C03628=1105.080,205.450,-68.281,178.823,14.144,151.208
C03629=1105.087,205.699,-68.305,178.828,14.143,151.207
C03630=1105.092,205.948,-68.330,178.832,14.142,151.206
C03631=1105.098,206.197,-68.354,178.836,14.141,151.205
C03632=1105.103,206.446,-68.379,178.840,14.139,151.203
C03633=1105.109,206.694,-68.403,178.845,14.138,151.202
C03634=1105.115,206.943,-68.427,178.848,14.136,151.201
C03635=1105.121,207.191,-68.452,178.853,14.136,151.200
C03636=1105.126,207.440,-68.476,178.857,14.134,151.198
C03637=1105.132,207.689,-68.501,178.861,14.133,151.197
C03638=1105.156,208.685,-68.598,178.887,14.133,151.191
C03639=1105.163,209.052,-68.635,178.893,14.132,151.190
C03640=1105.171,209.419,-68.670,178.899,14.131,151.188
C03641=1105.181,209.786,-68.707,178.904,14.131,151.187
C03642=1105.189,210.152,-68.743,178.911,14.131,151.186
C03643=1105.195,210.402,-68.768,178.914,14.129,151.185
C03644=1105.200,210.650,-68.792,178.918,14.129,151.184
C03645=1105.206,210.899,-68.817,178.922,14.129,151.183
C03646=1105.211,211.147,-68.841,178.926,14.129,151.182
C03647=1105.217,211.397,-68.866,178.930,14.128,151.181
C03648=1105.223,211.645,-68.891,178.934,14.127,151.180
C03649=1105.228,211.893,-68.915,178.938,14.127,151.179
C03650=1105.234,212.143,-68.940,178.942,14.126,151.178
C03651=1105.240,212.390,-68.965,178.946,14.126,151.177
C03652=1105.246,212.640,-68.990,178.949,14.125,151.176
C03653=1105.251,212.888,-69.014,178.953,14.125,151.175
C03654=1105.256,213.137,-69.040,178.958,14.125,151.174
C03655=1105.262,213.386,-69.064,178.961,14.125,151.173
C03656=1105.268,213.635,-69.089,178.966,14.124,151.172
C03657=1105.273,213.883,-69.114,178.969,14.123,151.171
C03658=1105.279,214.132,-69.139,178.973,14.123,151.170
C03659=1105.285,214.381,-69.164,178.977,14.123,151.169
C03660=1105.291,214.629,-69.188,178.981,14.122,151.168
C03661=1105.296,214.879,-69.214,178.985,14.122,151.167
C03662=1105.302,215.127,-69.239,178.989,14.122,151.166
C03663=1105.308,215.376,-69.263,178.993,14.121,151.165
C03664=1105.313,215.624,-69.288,178.997,14.120,151.164
C03665=1105.319,215.873,-69.313,179.001,14.120,151.163
C03666=1105.325,216.121,-69.338,179.005,14.120,151.162
C03667=1105.330,216.371,-69.363,179.009,14.119,151.161
C03668=1105.335,216.619,-69.388,179.012,14.119,151.160
C03669=1105.341,216.868,-69.413,179.017,14.118,151.159
C03670=1105.348,217.117,-69.438,179.020,14.118,151.158
C03671=1105.352,217.365,-69.464,179.025,14.118,151.157
C03672=1105.358,217.614,-69.488,179.029,14.118,151.156
C03673=1105.364,217.862,-69.513,179.033,14.117,151.155
C03674=1105.370,218.111,-69.539,179.036,14.116,151.154
C03675=1105.375,218.361,-69.564,179.040,14.116,151.153
C03676=1105.381,218.608,-69.589,179.044,14.116,151.152
C03677=1105.387,218.857,-69.614,179.048,14.115,151.151
C03678=1105.392,219.106,-69.638,179.052,14.115,151.150
C03679=1105.398,219.355,-69.664,179.056,14.115,151.149
C03680=1105.404,219.603,-69.690,179.060,14.114,151.148
C03681=1105.409,219.852,-69.714,179.064,14.114,151.147
C03682=1105.415,220.101,-69.740,179.068,14.113,151.146
C03683=1105.421,220.350,-69.765,179.072,14.113,151.145
C03684=1105.427,220.598,-69.790,179.076,14.113,151.144
C03685=1105.433,220.847,-69.815,179.080,14.112,151.143
C03686=1105.438,221.096,-69.841,179.083,14.112,151.142
C03687=1105.444,221.344,-69.866,179.087,14.111,151.141
C03688=1105.450,221.592,-69.891,179.092,14.111,151.140
C03689=1105.455,221.841,-69.917,179.096,14.111,151.139
C03690=1105.461,222.089,-69.942,179.100,14.110,151.138
C03691=1105.470,222.460,-69.980,179.105,14.110,151.137
C03692=1105.477,222.831,-70.017,179.111,14.109,151.135
C03693=1105.486,223.201,-70.056,179.117,14.108,151.134
C03694=1105.494,223.571,-70.093,179.123,14.108,151.133
C03695=1105.501,223.820,-70.119,179.127,14.108,151.132
C03696=1105.506,224.068,-70.144,179.131,14.107,151.131
C03697=1105.512,224.316,-70.169,179.134,14.107,151.130
C03698=1105.517,224.565,-70.195,179.139,14.107,151.129
C03699=1105.523,224.814,-70.221,179.143,14.107,151.128
C03700=1105.528,225.062,-70.246,179.147,14.106,151.127
C03701=1105.534,225.311,-70.272,179.151,14.106,151.126
C03702=1105.540,225.560,-70.298,179.155,14.106,151.125
C03703=1105.545,225.808,-70.323,179.159,14.106,151.124
C03704=1105.551,226.057,-70.348,179.162,14.105,151.123
C03705=1105.556,226.306,-70.374,179.166,14.104,151.122
C03706=1105.563,226.555,-70.400,179.170,14.104,151.121
C03707=1105.568,226.804,-70.426,179.174,14.104,151.120
C03708=1105.574,227.052,-70.451,179.178,14.104,151.119
C03709=1105.579,227.301,-70.477,179.182,14.103,151.118
C03710=1105.585,227.549,-70.502,179.186,14.103,151.117
C03711=1105.591,227.798,-70.528,179.191,14.103,151.116
C03712=1105.596,228.047,-70.553,179.194,14.102,151.115
C03713=1105.602,228.295,-70.579,179.198,14.102,151.114
C03714=1105.608,228.544,-70.605,179.202,14.102,151.113
C03715=1105.614,228.792,-70.631,179.206,14.102,151.112
C03716=1105.619,229.041,-70.657,179.210,14.101,151.111
C03717=1105.625,229.290,-70.683,179.214,14.101,151.110
C03718=1105.631,229.538,-70.708,179.218,14.101,151.109
C03719=1105.636,229.787,-70.734,179.222,14.101,151.108
C03720=1105.642,230.035,-70.760,179.226,14.100,151.107
C03721=1105.648,230.284,-70.785,179.229,14.100,151.107
C03722=1105.654,230.533,-70.812,179.234,14.099,151.105
C03723=1105.659,230.782,-70.838,179.237,14.099,151.105
C03724=1105.665,231.030,-70.863,179.241,14.099,151.104
C03725=1105.670,231.278,-70.889,179.246,14.099,151.103
C03726=1105.676,231.527,-70.916,179.250,14.099,151.102
C03727=1105.682,231.776,-70.942,179.254,14.098,151.101
C03728=1105.688,232.024,-70.967,179.258,14.098,151.100
C03729=1105.693,232.273,-70.994,179.262,14.098,151.099
C03730=1105.699,232.522,-71.019,179.266,14.098,151.098
C03731=1105.704,232.771,-71.045,179.269,14.097,151.097
C03732=1105.710,233.018,-71.072,179.273,14.097,151.096
C03733=1105.716,233.267,-71.097,179.277,14.097,151.095
C03734=1105.722,233.515,-71.124,179.281,14.096,151.094
C03735=1105.727,233.764,-71.150,179.285,14.096,151.093
C03736=1105.733,234.013,-71.175,179.289,14.096,151.092
C03737=1105.738,234.262,-71.202,179.293,14.096,151.091
C03738=1105.744,234.510,-71.227,179.297,14.096,151.090
C03739=1105.750,234.759,-71.254,179.301,14.096,151.089
C03740=1105.756,235.008,-71.280,179.305,14.096,151.089
C03741=1105.762,235.256,-71.307,179.309,14.095,151.087
C03742=1105.766,235.504,-71.332,179.313,14.095,151.087
C03743=1105.775,235.867,-71.371,179.319,14.094,151.085
C03744=1105.783,236.228,-71.409,179.324,14.094,151.084
C03745=1105.791,236.590,-71.448,179.330,14.094,151.083
C03746=1105.799,236.952,-71.486,179.336,14.094,151.081
C03747=1105.805,237.201,-71.512,179.340,14.094,151.080
C03748=1105.810,237.449,-71.539,179.344,14.093,151.079
C03749=1105.816,237.698,-71.564,179.348,14.093,151.078
C03750=1105.822,237.946,-71.591,179.351,14.093,151.077
C03751=1105.828,238.194,-71.617,179.355,14.092,151.076
C03752=1105.834,238.443,-71.643,179.359,14.092,151.075
C03753=1105.839,238.692,-71.670,179.363,14.092,151.075
C03754=1105.845,238.940,-71.696,179.367,14.092,151.074
C03755=1105.851,239.189,-71.722,179.371,14.092,151.073
C03756=1105.856,239.437,-71.749,179.375,14.092,151.072
C03757=1105.862,239.686,-71.776,179.379,14.091,151.071
C03758=1105.868,239.935,-71.802,179.383,14.091,151.070
C03759=1105.874,240.183,-71.828,179.387,14.091,151.069
C03760=1105.879,240.432,-71.855,179.391,14.091,151.068
C03761=1105.884,240.680,-71.882,179.395,14.091,151.067
C03762=1105.890,240.929,-71.908,179.399,14.091,151.066
C03763=1105.896,241.178,-71.935,179.403,14.091,151.065
C03764=1105.902,241.426,-71.962,179.407,14.090,151.064
C03765=1105.908,241.675,-71.988,179.411,14.090,151.063
C03766=1105.913,241.923,-72.015,179.415,14.090,151.062
C03767=1105.919,242.172,-72.042,179.419,14.090,151.061
C03768=1105.925,242.420,-72.068,179.423,14.090,151.060
C03769=1105.931,242.669,-72.094,179.427,14.090,151.060
C03770=1105.936,242.917,-72.121,179.431,14.090,151.059
C03771=1105.942,243.166,-72.147,179.435,14.090,151.058
C03772=1105.947,243.414,-72.175,179.439,14.090,151.057
C03773=1105.953,243.663,-72.201,179.443,14.090,151.056
C03774=1105.959,243.911,-72.228,179.446,14.089,151.055
C03775=1105.964,244.159,-72.255,179.450,14.089,151.054
C03776=1105.970,244.409,-72.282,179.454,14.089,151.053
C03777=1105.976,244.657,-72.309,179.458,14.089,151.052
C03778=1105.982,244.905,-72.336,179.462,14.089,151.051
C03779=1105.987,245.154,-72.362,179.466,14.089,151.050
C03780=1105.992,245.402,-72.389,179.470,14.088,151.049
C03781=1105.998,245.651,-72.416,179.474,14.088,151.049
C03782=1106.004,245.899,-72.443,179.478,14.088,151.048
C03783=1106.010,246.148,-72.469,179.482,14.088,151.047
C03784=1106.015,246.396,-72.497,179.486,14.088,151.046
C03785=1106.021,246.645,-72.524,179.490,14.088,151.045
C03786=1106.027,246.894,-72.550,179.494,14.088,151.044
C03787=1106.032,247.142,-72.578,179.498,14.088,151.043
C03788=1106.038,247.391,-72.604,179.501,14.088,151.042
C03789=1106.043,247.639,-72.631,179.505,14.088,151.041
C03790=1106.049,247.888,-72.658,179.510,14.087,151.040
C03791=1106.055,248.135,-72.685,179.513,14.087,151.039
C03792=1106.060,248.384,-72.712,179.517,14.087,151.039
C03793=1106.066,248.633,-72.740,179.521,14.087,151.038
C03794=1106.072,248.882,-72.766,179.525,14.087,151.037
C03795=1106.079,249.237,-72.805,179.531,14.088,151.036
C03796=1106.087,249.591,-72.844,179.537,14.087,151.034
C03797=1106.095,249.947,-72.883,179.542,14.087,151.033
C03798=1106.104,250.302,-72.921,179.548,14.088,151.032
C03799=1106.109,250.550,-72.949,179.552,14.088,151.031
C03800=1106.115,250.799,-72.976,179.556,14.088,151.030
C03801=1106.120,251.047,-73.003,179.560,14.088,151.029
C03802=1106.127,251.296,-73.031,179.564,14.088,151.028
C03803=1106.132,251.544,-73.058,179.568,14.088,151.027
C03804=1106.137,251.793,-73.085,179.572,14.088,151.026
C03805=1106.143,252.041,-73.112,179.576,14.088,151.025
C03806=1106.149,252.290,-73.139,179.579,14.088,151.025
C03807=1106.154,252.539,-73.167,179.583,14.088,151.024
C03808=1106.159,252.787,-73.195,179.587,14.088,151.023
C03809=1106.165,253.035,-73.221,179.591,14.088,151.022
C03810=1106.170,253.284,-73.249,179.595,14.088,151.021
C03811=1106.177,253.532,-73.276,179.599,14.088,151.020
C03812=1106.182,253.781,-73.304,179.603,14.088,151.019
C03813=1106.188,254.028,-73.331,179.607,14.088,151.018
C03814=1106.194,254.278,-73.359,179.611,14.088,151.018
C03815=1106.200,254.526,-73.386,179.614,14.088,151.017
C03816=1106.205,254.774,-73.413,179.619,14.087,151.016
C03817=1106.210,255.022,-73.441,179.623,14.088,151.015
C03818=1106.217,255.271,-73.468,179.627,14.088,151.014
C03819=1106.222,255.519,-73.496,179.631,14.088,151.013
C03820=1106.228,255.768,-73.523,179.635,14.088,151.012
C03821=1106.234,256.017,-73.551,179.639,14.088,151.011
C03822=1106.239,256.265,-73.578,179.643,14.088,151.010
C03823=1106.245,256.513,-73.606,179.647,14.088,151.009
C03824=1106.251,256.762,-73.634,179.650,14.088,151.009
C03825=1106.256,257.010,-73.661,179.654,14.088,151.008
C03826=1106.262,257.258,-73.689,179.658,14.088,151.007
C03827=1106.267,257.507,-73.716,179.662,14.088,151.006
C03828=1106.273,257.756,-73.744,179.666,14.088,151.005
C03829=1106.279,258.003,-73.772,179.670,14.088,151.004
C03830=1106.284,258.253,-73.799,179.674,14.088,151.003
C03831=1106.290,258.501,-73.827,179.678,14.089,151.003
C03832=1106.296,258.749,-73.855,179.681,14.089,151.002
C03833=1106.302,258.997,-73.883,179.685,14.089,151.001
C03834=1106.307,259.246,-73.910,179.690,14.089,151.000
C03835=1106.314,259.494,-73.938,179.694,14.089,150.999
C03836=1106.319,259.742,-73.966,179.698,14.089,150.998
C03837=1106.325,259.991,-73.994,179.702,14.089,150.997
C03838=1106.331,260.239,-74.021,179.706,14.089,150.996
C03839=1106.336,260.487,-74.049,179.710,14.089,150.995
C03840=1106.342,260.736,-74.077,179.714,14.089,150.995
C03841=1106.347,260.984,-74.105,179.717,14.089,150.994
C03842=1106.354,261.233,-74.133,179.721,14.089,150.993
C03843=1106.359,261.481,-74.160,179.725,14.089,150.992
C03844=1106.365,261.730,-74.188,179.729,14.089,150.991
C03845=1106.370,261.978,-74.216,179.733,14.089,150.990
C03846=1106.377,262.227,-74.244,179.737,14.089,150.989
C03847=1106.385,262.579,-74.284,179.743,14.090,150.988
C03848=1106.393,262.931,-74.324,179.748,14.090,150.987
C03849=1106.400,263.284,-74.363,179.754,14.091,150.986
C03850=1106.409,263.636,-74.403,179.759,14.090,150.984
C03851=1106.414,263.885,-74.431,179.763,14.090,150.984
C03852=1106.421,264.133,-74.459,179.767,14.091,150.983
C03853=1106.426,264.381,-74.487,179.771,14.091,150.982
C03854=1106.432,264.630,-74.515,179.775,14.091,150.981
C03855=1106.438,264.878,-74.543,179.779,14.091,150.980
C03856=1106.444,265.127,-74.571,179.783,14.091,150.979
C03857=1106.449,265.375,-74.599,179.787,14.092,150.979
C03858=1106.455,265.623,-74.627,179.791,14.092,150.978
C03859=1106.460,265.871,-74.655,179.795,14.092,150.977
C03860=1106.466,266.120,-74.684,179.798,14.092,150.976
C03861=1106.472,266.368,-74.712,179.802,14.092,150.975
C03862=1106.478,266.616,-74.741,179.806,14.092,150.974
C03863=1106.483,266.864,-74.769,179.810,14.093,150.973
C03864=1106.489,267.113,-74.797,179.814,14.093,150.973
C03865=1106.494,267.361,-74.825,179.818,14.093,150.972
C03866=1106.500,267.610,-74.853,179.822,14.093,150.971
C03867=1106.506,267.857,-74.882,179.826,14.093,150.970
C03868=1106.512,268.106,-74.910,179.830,14.094,150.969
C03869=1106.517,268.354,-74.938,179.833,14.094,150.968
C03870=1106.523,268.603,-74.967,179.837,14.094,150.968
C03871=1106.529,268.852,-74.995,179.842,14.095,150.967
C03872=1106.535,269.099,-75.024,179.846,14.095,150.966
C03873=1106.540,269.348,-75.053,179.850,14.095,150.965
C03874=1106.545,269.596,-75.080,179.853,14.095,150.964
C03875=1106.551,269.845,-75.109,179.857,14.095,150.963
C03876=1106.557,270.092,-75.137,179.861,14.095,150.963
C03877=1106.563,270.341,-75.166,179.865,14.096,150.962
C03878=1106.569,270.590,-75.194,179.869,14.097,150.961
C03879=1106.574,270.837,-75.223,179.873,14.097,150.960
C03880=1106.580,271.086,-75.252,179.877,14.097,150.959
C03881=1106.585,271.334,-75.280,179.881,14.097,150.958
C03882=1106.591,271.583,-75.309,179.884,14.097,150.958
C03883=1106.597,271.831,-75.337,179.888,14.097,150.957
C03884=1106.603,272.079,-75.366,179.892,14.097,150.956
C03885=1106.608,272.328,-75.395,179.896,14.099,150.955
C03886=1106.613,272.576,-75.423,179.900,14.099,150.954
C03887=1106.620,272.824,-75.452,179.904,14.099,150.954
C03888=1106.626,273.073,-75.480,179.907,14.099,150.953
C03889=1106.631,273.320,-75.509,179.911,14.099,150.952
C03890=1106.636,273.569,-75.538,179.915,14.099,150.951
C03891=1106.643,273.817,-75.567,179.920,14.100,150.950
C03892=1106.648,274.065,-75.595,179.923,14.101,150.950
C03893=1106.654,274.314,-75.624,179.927,14.101,150.949
C03894=1106.659,274.562,-75.652,179.931,14.101,150.948
C03895=1106.665,274.810,-75.681,179.935,14.101,150.947
C03896=1106.671,275.059,-75.710,179.939,14.102,150.946
C03897=1106.676,275.307,-75.739,179.943,14.102,150.946
C03898=1106.682,275.555,-75.768,179.947,14.103,150.945
C03899=1106.690,275.910,-75.809,179.952,14.102,150.944
C03900=1106.698,276.266,-75.851,179.957,14.104,150.943
C03901=1106.707,276.621,-75.891,179.963,14.104,150.941
C03902=1106.715,276.976,-75.933,179.968,14.105,150.940
C03903=1106.720,277.224,-75.962,179.972,14.105,150.939
C03904=1106.726,277.473,-75.990,179.977,14.106,150.939
C03905=1106.732,277.721,-76.020,179.980,14.106,150.938
C03906=1106.737,277.970,-76.049,179.984,14.106,150.937
C03907=1106.743,278.217,-76.078,179.988,14.106,150.936
C03908=1106.748,278.466,-76.107,179.992,14.107,150.936
C03909=1106.755,278.714,-76.136,179.996,14.108,150.935
C03910=1106.759,278.962,-76.165,180.000,14.108,150.934
C03911=1106.766,279.210,-76.194,-179.997,14.108,150.933
C03912=1106.771,279.459,-76.223,-179.993,14.108,150.932
C03913=1106.777,279.707,-76.252,-179.989,14.109,150.932
C03914=1106.782,279.955,-76.281,-179.985,14.110,150.931
C03915=1106.788,280.203,-76.310,-179.981,14.110,150.930
C03916=1106.794,280.452,-76.340,-179.977,14.110,150.929
C03917=1106.800,280.700,-76.369,-179.974,14.111,150.929
C03918=1106.806,280.948,-76.399,-179.969,14.111,150.928
C03919=1106.811,281.196,-76.427,-179.966,14.112,150.927
C03920=1106.816,281.445,-76.456,-179.962,14.112,150.926
C03921=1106.823,281.693,-76.485,-179.958,14.112,150.926
C03922=1106.828,281.941,-76.515,-179.955,14.113,150.925
C03923=1106.834,282.189,-76.544,-179.950,14.114,150.924
C03924=1106.839,282.437,-76.573,-179.947,14.114,150.923
C03925=1106.845,282.685,-76.603,-179.943,14.114,150.923
C03926=1106.851,282.934,-76.632,-179.939,14.115,150.922
C03927=1106.856,283.181,-76.661,-179.935,14.116,150.921
C03928=1106.862,283.430,-76.691,-179.931,14.116,150.920
C03929=1106.868,283.678,-76.720,-179.928,14.117,150.920
C03930=1106.873,283.926,-76.750,-179.924,14.117,150.919
C03931=1106.879,284.175,-76.779,-179.919,14.118,150.918
C03932=1106.885,284.423,-76.808,-179.916,14.118,150.917
C03933=1106.890,284.671,-76.837,-179.912,14.118,150.917
C03934=1106.896,284.919,-76.867,-179.909,14.119,150.916
C03935=1106.902,285.167,-76.896,-179.904,14.120,150.915
C03936=1106.908,285.415,-76.926,-179.900,14.120,150.914
C03937=1106.913,285.664,-76.956,-179.897,14.121,150.914
C03938=1106.919,285.912,-76.986,-179.893,14.122,150.913
C03939=1106.924,286.159,-77.014,-179.889,14.122,150.912
C03940=1106.930,286.408,-77.044,-179.885,14.122,150.911
C03941=1106.935,286.656,-77.074,-179.882,14.123,150.911
C03942=1106.942,286.904,-77.103,-179.878,14.124,150.910
C03943=1106.947,287.152,-77.133,-179.874,14.124,150.909
C03944=1106.953,287.401,-77.163,-179.870,14.125,150.909
C03945=1106.958,287.649,-77.192,-179.867,14.125,150.908
C03946=1106.965,287.897,-77.221,-179.862,14.126,150.907
C03947=1106.970,288.145,-77.252,-179.859,14.126,150.906
C03948=1106.975,288.393,-77.281,-179.855,14.127,150.906
C03949=1106.981,288.641,-77.311,-179.850,14.128,150.905
C03950=1106.987,288.889,-77.341,-179.847,14.128,150.904
C03951=1106.996,289.254,-77.384,-179.841,14.129,150.903
C03952=1107.005,289.619,-77.428,-179.836,14.130,150.902
C03953=1107.013,289.983,-77.472,-179.830,14.130,150.901
C03954=1107.020,290.348,-77.516,-179.825,14.132,150.900
C03955=1107.027,290.596,-77.545,-179.821,14.132,150.899
C03956=1107.032,290.845,-77.575,-179.817,14.133,150.899
C03957=1107.038,291.093,-77.605,-179.813,14.134,150.898
C03958=1107.043,291.341,-77.635,-179.810,14.134,150.897
C03959=1107.049,291.589,-77.665,-179.806,14.135,150.896
C03960=1107.055,291.837,-77.695,-179.802,14.136,150.896
C03961=1107.061,292.085,-77.725,-179.798,14.136,150.895
C03962=1107.066,292.334,-77.755,-179.794,14.137,150.894
C03963=1107.072,292.581,-77.785,-179.791,14.138,150.894
C03964=1107.077,292.830,-77.815,-179.787,14.138,150.893
C03965=1107.083,293.078,-77.845,-179.783,14.139,150.892
C03966=1107.089,293.326,-77.875,-179.779,14.140,150.892
C03967=1107.095,293.574,-77.905,-179.776,14.140,150.891
C03968=1107.100,293.822,-77.935,-179.771,14.142,150.890
C03969=1107.106,294.070,-77.965,-179.768,14.142,150.890
C03970=1107.112,294.318,-77.995,-179.764,14.143,150.889
C03971=1107.117,294.567,-78.025,-179.760,14.144,150.888
C03972=1107.123,294.814,-78.055,-179.756,14.144,150.887
C03973=1107.129,295.062,-78.086,-179.753,14.145,150.887
C03974=1107.134,295.311,-78.115,-179.749,14.146,150.886
C03975=1107.140,295.558,-78.146,-179.745,14.146,150.885
C03976=1107.146,295.806,-78.176,-179.742,14.147,150.885
C03977=1107.152,296.055,-78.206,-179.737,14.148,150.884
C03978=1107.157,296.303,-78.236,-179.734,14.148,150.883
C03979=1107.162,296.551,-78.267,-179.730,14.149,150.883
C03980=1107.168,296.799,-78.297,-179.726,14.150,150.882
C03981=1107.174,297.047,-78.327,-179.723,14.151,150.881
C03982=1107.180,297.295,-78.357,-179.719,14.152,150.881
C03983=1107.185,297.543,-78.388,-179.715,14.153,150.880
C03984=1107.191,297.790,-78.418,-179.712,14.153,150.879
C03985=1107.197,298.039,-78.448,-179.707,14.155,150.879
C03986=1107.202,298.287,-78.479,-179.704,14.155,150.878
C03987=1107.208,298.535,-78.509,-179.700,14.156,150.877
C03988=1107.214,298.783,-78.540,-179.696,14.157,150.877
C03989=1107.220,299.031,-78.570,-179.693,14.157,150.876
C03990=1107.225,299.280,-78.600,-179.689,14.159,150.876
C03991=1107.230,299.528,-78.631,-179.685,14.159,150.875
C03992=1107.236,299.776,-78.661,-179.682,14.160,150.874
C03993=1107.241,300.024,-78.692,-179.677,14.161,150.874
C03994=1107.247,300.271,-78.722,-179.674,14.162,150.873
C03995=1107.253,300.519,-78.753,-179.670,14.163,150.872
C03996=1107.258,300.767,-78.784,-179.666,14.164,150.872
C03997=1107.264,301.015,-78.814,-179.663,14.164,150.871
C03998=1107.270,301.263,-78.844,-179.659,14.166,150.871
C03999=1107.275,301.511,-78.875,-179.656,14.166,150.870
C04000=1107.281,301.759,-78.906,-179.651,14.168,150.869
C04001=1107.286,302.007,-78.937,-179.648,14.168,150.869
C04002=1107.292,302.256,-78.967,-179.645,14.169,150.868
C04003=1107.300,302.634,-79.013,-179.638,14.171,150.867
C04004=1107.309,303.013,-79.061,-179.633,14.172,150.866
C04005=1107.318,303.391,-79.108,-179.627,14.174,150.865
C04006=1107.326,303.770,-79.154,-179.622,14.175,150.864
C04007=1107.331,304.018,-79.185,-179.618,14.176,150.864
C04008=1107.337,304.266,-79.215,-179.614,14.177,150.863
C04009=1107.343,304.514,-79.247,-179.610,14.178,150.862
C04010=1107.349,304.762,-79.278,-179.607,14.179,150.862
C04011=1107.355,305.010,-79.308,-179.603,14.180,150.861
C04012=1107.360,305.258,-79.339,-179.599,14.181,150.861
C04013=1107.366,305.506,-79.369,-179.595,14.182,150.860
C04014=1107.372,305.754,-79.402,-179.592,14.183,150.859
C04015=1107.378,306.002,-79.432,-179.589,14.184,150.859
C04016=1107.383,306.250,-79.463,-179.584,14.185,150.858
C04017=1107.389,306.498,-79.493,-179.581,14.185,150.858
C04018=1107.394,306.745,-79.525,-179.577,14.187,150.857
C04019=1107.400,306.994,-79.556,-179.573,14.188,150.856
C04020=1107.405,307.242,-79.586,-179.570,14.189,150.856
C04021=1107.412,307.489,-79.618,-179.566,14.190,150.855
C04022=1107.417,307.737,-79.648,-179.562,14.191,150.855
C04023=1107.423,307.986,-79.679,-179.559,14.192,150.854
C04024=1107.428,308.233,-79.711,-179.555,14.194,150.854
C04025=1107.433,308.482,-79.742,-179.551,14.194,150.853
C04026=1107.440,308.730,-79.773,-179.547,14.195,150.852
C04027=1107.445,308.978,-79.804,-179.544,14.196,150.852
C04028=1107.451,309.225,-79.835,-179.540,14.197,150.851
C04029=1107.457,309.474,-79.867,-179.536,14.198,150.851
C04030=1107.463,309.721,-79.897,-179.533,14.199,150.850
C04031=1107.468,309.970,-79.928,-179.529,14.201,150.849
C04032=1107.474,310.218,-79.960,-179.526,14.201,150.849
C04033=1107.480,310.466,-79.990,-179.522,14.203,150.848
C04034=1107.485,310.713,-80.022,-179.518,14.204,150.848
C04035=1107.492,310.962,-80.053,-179.514,14.205,150.847
C04036=1107.497,311.209,-80.084,-179.511,14.206,150.847
C04037=1107.502,311.457,-80.115,-179.507,14.207,150.846
C04038=1107.509,311.705,-80.147,-179.504,14.208,150.845
C04039=1107.514,311.953,-80.178,-179.499,14.209,150.845
C04040=1107.520,312.202,-80.210,-179.496,14.210,150.844
C04041=1107.526,312.449,-80.241,-179.492,14.212,150.844
C04042=1107.531,312.697,-80.272,-179.489,14.212,150.843
C04043=1107.537,312.945,-80.304,-179.485,14.214,150.843
C04044=1107.543,313.192,-80.335,-179.481,14.214,150.842
C04045=1107.549,313.441,-80.366,-179.478,14.216,150.842
C04046=1107.554,313.689,-80.398,-179.474,14.217,150.841
C04047=1107.561,313.937,-80.429,-179.470,14.218,150.840
C04048=1107.566,314.185,-80.460,-179.467,14.219,150.840
C04049=1107.571,314.432,-80.492,-179.463,14.221,150.839
C04050=1107.577,314.680,-80.524,-179.460,14.221,150.839
C04051=1107.583,314.928,-80.554,-179.456,14.223,150.838
C04052=1107.589,315.176,-80.586,-179.453,14.224,150.838
C04053=1107.595,315.424,-80.618,-179.449,14.226,150.837
C04054=1107.601,315.672,-80.650,-179.445,14.226,150.837
C04055=1107.609,316.053,-80.698,-179.440,14.229,150.836
C04056=1107.617,316.434,-80.747,-179.434,14.230,150.835
C04057=1107.626,316.816,-80.795,-179.428,14.233,150.834
C04058=1107.634,317.197,-80.844,-179.423,14.234,150.834
C04059=1107.640,317.445,-80.875,-179.419,14.236,150.833
C04060=1107.646,317.693,-80.907,-179.416,14.237,150.833
C04061=1107.651,317.941,-80.939,-179.412,14.239,150.832
C04062=1107.657,318.189,-80.971,-179.409,14.240,150.832
C04063=1107.662,318.436,-81.003,-179.405,14.241,150.831
C04064=1107.668,318.685,-81.035,-179.401,14.243,150.831
C04065=1107.674,318.932,-81.066,-179.398,14.244,150.830
C04066=1107.680,319.181,-81.098,-179.394,14.245,150.830
C04067=1107.685,319.428,-81.129,-179.391,14.246,150.829
C04068=1107.691,319.677,-81.161,-179.387,14.248,150.829
C04069=1107.696,319.924,-81.193,-179.383,14.250,150.828
C04070=1107.702,320.172,-81.225,-179.380,14.251,150.828
C04071=1107.708,320.420,-81.257,-179.376,14.252,150.827
C04072=1107.714,320.668,-81.289,-179.374,14.254,150.827
C04073=1107.718,320.916,-81.321,-179.370,14.255,150.827
C04074=1107.724,321.164,-81.353,-179.367,14.256,150.826
C04075=1107.730,321.412,-81.385,-179.363,14.258,150.826
C04076=1107.736,321.659,-81.418,-179.359,14.259,150.825
C04077=1107.741,321.907,-81.449,-179.356,14.260,150.825
C04078=1107.747,322.155,-81.481,-179.352,14.262,150.824
C04079=1107.753,322.403,-81.513,-179.349,14.263,150.824
C04080=1107.759,322.651,-81.545,-179.345,14.265,150.823
C04081=1107.764,322.899,-81.578,-179.341,14.267,150.823
C04082=1107.769,323.147,-81.609,-179.338,14.268,150.822
C04083=1107.775,323.395,-81.641,-179.334,14.269,150.822
C04084=1107.781,323.642,-81.674,-179.331,14.271,150.822
C04085=1107.787,323.890,-81.706,-179.327,14.272,150.821
C04086=1107.793,324.138,-81.738,-179.324,14.274,150.821
C04087=1107.798,324.386,-81.770,-179.320,14.275,150.820
C04088=1107.804,324.634,-81.802,-179.317,14.277,150.820
C04089=1107.810,324.882,-81.835,-179.313,14.278,150.819
C04090=1107.815,325.129,-81.866,-179.310,14.279,150.819
C04091=1107.821,325.378,-81.899,-179.306,14.281,150.818
C04092=1107.826,325.626,-81.931,-179.302,14.283,150.818
C04093=1107.832,325.873,-81.963,-179.299,14.284,150.818
C04094=1107.838,326.121,-81.995,-179.295,14.286,150.817
C04095=1107.844,326.369,-82.027,-179.292,14.288,150.817
C04096=1107.849,326.617,-82.060,-179.289,14.289,150.816
C04097=1107.855,326.865,-82.092,-179.285,14.290,150.816
C04098=1107.861,327.113,-82.124,-179.282,14.292,150.816
C04099=1107.866,327.360,-82.157,-179.278,14.293,150.815
C04100=1107.872,327.609,-82.189,-179.274,14.295,150.815
C04101=1107.878,327.856,-82.222,-179.271,14.296,150.814
C04102=1107.884,328.104,-82.254,-179.267,14.298,150.814
C04103=1107.889,328.352,-82.287,-179.264,14.300,150.814
C04104=1107.895,328.600,-82.319,-179.261,14.301,150.813
C04105=1107.901,328.848,-82.351,-179.257,14.303,150.813
C04106=1107.906,329.095,-82.384,-179.253,14.304,150.812
C04107=1107.915,329.470,-82.434,-179.248,14.306,150.812
C04108=1107.923,329.844,-82.482,-179.243,14.309,150.811
C04109=1107.932,330.218,-82.532,-179.237,14.312,150.811
C04110=1107.942,330.592,-82.581,-179.233,14.314,150.810
C04111=1107.947,330.840,-82.613,-179.229,14.316,150.810
C04112=1107.953,331.088,-82.645,-179.225,14.318,150.809
C04113=1107.959,331.336,-82.679,-179.222,14.319,150.809
C04114=1107.964,331.584,-82.711,-179.218,14.321,150.808
C04115=1107.971,331.831,-82.744,-179.215,14.323,150.808
C04116=1107.976,332.079,-82.777,-179.212,14.324,150.808
C04117=1107.982,332.327,-82.809,-179.208,14.326,150.807
C04118=1107.987,332.575,-82.842,-179.205,14.328,150.807
C04119=1107.994,332.822,-82.875,-179.201,14.330,150.807
C04120=1107.999,333.071,-82.907,-179.198,14.331,150.806
C04121=1108.004,333.318,-82.940,-179.194,14.333,150.806
C04122=1108.010,333.566,-82.973,-179.191,14.335,150.806
C04123=1108.016,333.814,-83.006,-179.187,14.337,150.805
C04124=1108.022,334.062,-83.038,-179.184,14.338,150.805
C04125=1108.027,334.310,-83.072,-179.181,14.340,150.805
C04126=1108.032,334.557,-83.105,-179.177,14.342,150.804
C04127=1108.038,334.805,-83.137,-179.174,14.344,150.804
C04128=1108.044,335.052,-83.171,-179.171,14.345,150.804
C04129=1108.050,335.301,-83.203,-179.167,14.347,150.803
C04130=1108.056,335.549,-83.236,-179.164,14.349,150.803
C04131=1108.060,335.796,-83.269,-179.160,14.351,150.803
C04132=1108.067,336.043,-83.302,-179.157,14.352,150.802
C04133=1108.072,336.291,-83.335,-179.153,14.354,150.802
C04134=1108.078,336.539,-83.369,-179.150,14.357,150.802
C04135=1108.084,336.787,-83.401,-179.146,14.359,150.801
C04136=1108.089,337.035,-83.434,-179.143,14.361,150.801
C04137=1108.095,337.283,-83.467,-179.140,14.362,150.801
C04138=1108.101,337.531,-83.500,-179.136,14.364,150.801
C04139=1108.106,337.778,-83.533,-179.133,14.366,150.800
C04140=1108.112,338.026,-83.566,-179.129,14.368,150.800
C04141=1108.117,338.274,-83.600,-179.126,14.370,150.800
C04142=1108.124,338.521,-83.632,-179.123,14.371,150.799
C04143=1108.129,338.769,-83.666,-179.120,14.373,150.799
C04144=1108.135,339.017,-83.699,-179.116,14.376,150.799
C04145=1108.140,339.265,-83.732,-179.113,14.378,150.799
C04146=1108.147,339.512,-83.766,-179.109,14.380,150.798
C04147=1108.152,339.760,-83.799,-179.106,14.382,150.798
C04148=1108.158,340.008,-83.833,-179.103,14.383,150.798
C04149=1108.163,340.255,-83.865,-179.099,14.385,150.797
C04150=1108.168,340.503,-83.899,-179.096,14.388,150.797
C04151=1108.174,340.751,-83.932,-179.093,14.390,150.797
C04152=1108.180,340.999,-83.965,-179.089,14.392,150.797
C04153=1108.186,341.246,-83.998,-179.086,14.394,150.796
C04154=1108.191,341.494,-84.032,-179.082,14.396,150.796
C04155=1108.197,341.742,-84.066,-179.080,14.398,150.796
C04156=1108.203,341.989,-84.099,-179.076,14.400,150.796
C04157=1108.208,342.237,-84.132,-179.073,14.402,150.796
C04158=1108.214,342.485,-84.166,-179.069,14.404,150.795
C04159=1108.223,342.853,-84.215,-179.064,14.408,150.795
C04160=1108.231,343.221,-84.265,-179.059,14.411,150.795
C04161=1108.240,343.589,-84.315,-179.055,14.414,150.794
C04162=1108.248,343.957,-84.364,-179.049,14.417,150.794
C04163=1108.254,344.205,-84.399,-179.046,14.419,150.794
C04164=1108.259,344.453,-84.432,-179.043,14.421,150.793
C04165=1108.265,344.700,-84.465,-179.040,14.424,150.793
C04166=1108.271,344.948,-84.499,-179.036,14.426,150.793
C04167=1108.276,345.196,-84.533,-179.033,14.428,150.793
C04168=1108.282,345.443,-84.567,-179.029,14.430,150.793
C04169=1108.288,345.691,-84.600,-179.026,14.432,150.793
C04170=1108.293,345.939,-84.633,-179.023,14.434,150.792
C04171=1108.299,346.186,-84.667,-179.020,14.436,150.792
C04172=1108.305,346.434,-84.701,-179.017,14.439,150.792
C04173=1108.311,346.681,-84.735,-179.013,14.441,150.792
C04174=1108.316,346.929,-84.768,-179.010,14.443,150.792
C04175=1108.321,347.177,-84.803,-179.007,14.446,150.791
C04176=1108.327,347.425,-84.836,-179.003,14.448,150.791
C04177=1108.333,347.672,-84.870,-179.000,14.450,150.791
C04178=1108.338,347.920,-84.904,-178.997,14.452,150.791
C04179=1108.345,348.168,-84.938,-178.994,14.455,150.791
C04180=1108.350,348.416,-84.971,-178.990,14.457,150.791
C04181=1108.356,348.663,-85.005,-178.987,14.459,150.790
C04182=1108.361,348.911,-85.040,-178.984,14.462,150.790
C04183=1108.367,349.158,-85.073,-178.981,14.464,150.790
C04184=1108.373,349.406,-85.107,-178.978,14.467,150.790
C04185=1108.378,349.653,-85.141,-178.974,14.469,150.790
C04186=1108.384,349.901,-85.175,-178.971,14.471,150.790
C04187=1108.390,350.148,-85.209,-178.968,14.474,150.790
C04188=1108.395,350.396,-85.243,-178.964,14.476,150.789
C04189=1108.401,350.644,-85.277,-178.961,14.478,150.789
C04190=1108.406,350.891,-85.311,-178.958,14.481,150.789
C04191=1108.413,351.139,-85.345,-178.955,14.483,150.789
C04192=1108.418,351.387,-85.379,-178.952,14.486,150.789
C04193=1108.424,351.634,-85.413,-178.948,14.488,150.789
C04194=1108.429,351.882,-85.447,-178.945,14.491,150.789
C04195=1108.435,352.129,-85.481,-178.942,14.493,150.789
C04196=1108.440,352.377,-85.516,-178.939,14.495,150.789
C04197=1108.446,352.625,-85.549,-178.936,14.498,150.788
C04198=1108.452,352.873,-85.584,-178.932,14.500,150.788
C04199=1108.458,353.120,-85.618,-178.929,14.503,150.788
C04200=1108.463,353.367,-85.652,-178.926,14.505,150.788
C04201=1108.469,353.615,-85.686,-178.923,14.508,150.788
C04202=1108.474,353.862,-85.721,-178.920,14.510,150.788
C04203=1108.480,354.110,-85.755,-178.917,14.513,150.788
C04204=1108.486,354.358,-85.789,-178.914,14.515,150.788
C04205=1108.492,354.606,-85.824,-178.911,14.518,150.788
C04206=1108.497,354.853,-85.858,-178.908,14.521,150.788
C04207=1108.503,355.101,-85.892,-178.904,14.523,150.788
C04208=1108.508,355.348,-85.926,-178.901,14.525,150.787
C04209=1108.513,355.596,-85.961,-178.898,14.529,150.788
C04210=1108.520,355.844,-85.995,-178.894,14.531,150.787
C04211=1108.528,356.213,-86.046,-178.890,14.535,150.787
C04212=1108.538,356.583,-86.099,-178.885,14.539,150.787
C04213=1108.545,356.954,-86.150,-178.881,14.543,150.787
C04214=1108.554,357.323,-86.201,-178.876,14.547,150.787
C04215=1108.559,357.572,-86.236,-178.873,14.550,150.787
C04216=1108.565,357.819,-86.270,-178.870,14.552,150.787
C04217=1108.570,358.067,-86.305,-178.867,14.555,150.787
C04218=1108.576,358.314,-86.339,-178.863,14.558,150.787
C04219=1108.582,358.562,-86.375,-178.860,14.561,150.787
C04220=1108.588,358.809,-86.409,-178.857,14.564,150.787
C04221=1108.593,359.057,-86.444,-178.854,14.566,150.787
C04222=1108.599,359.304,-86.478,-178.851,14.569,150.787
C04223=1108.605,359.552,-86.513,-178.849,14.572,150.787
C04224=1108.611,359.799,-86.547,-178.845,14.574,150.787
C04225=1108.616,360.046,-86.582,-178.842,14.577,150.787
C04226=1108.622,360.294,-86.616,-178.839,14.580,150.787
C04227=1108.628,360.541,-86.652,-178.836,14.583,150.787
C04228=1108.633,360.789,-86.686,-178.833,14.586,150.787
C04229=1108.639,361.036,-86.720,-178.830,14.588,150.787
C04230=1108.645,361.284,-86.756,-178.827,14.591,150.787
C04231=1108.650,361.531,-86.791,-178.824,14.594,150.787
C04232=1108.656,361.779,-86.825,-178.821,14.596,150.787
C04233=1108.662,362.026,-86.861,-178.817,14.600,150.787
C04234=1108.667,362.274,-86.895,-178.815,14.603,150.787
C04235=1108.673,362.521,-86.929,-178.812,14.606,150.787
C04236=1108.679,362.769,-86.965,-178.809,14.608,150.787
C04237=1108.684,363.017,-87.000,-178.806,14.611,150.787
C04238=1108.689,363.264,-87.035,-178.802,14.615,150.788
C04239=1108.696,363.512,-87.070,-178.800,14.618,150.788
C04240=1108.701,363.758,-87.105,-178.797,14.620,150.788
C04241=1108.706,364.006,-87.140,-178.794,14.623,150.788
C04242=1108.713,364.253,-87.175,-178.791,14.626,150.788
C04243=1108.718,364.501,-87.209,-178.787,14.630,150.788
C04244=1108.724,364.748,-87.245,-178.785,14.632,150.788
C04245=1108.730,364.996,-87.280,-178.782,14.635,150.788
C04246=1108.735,365.243,-87.315,-178.779,14.638,150.788
C04247=1108.741,365.491,-87.349,-178.776,14.641,150.788
C04248=1108.747,365.738,-87.385,-178.773,14.645,150.788
C04249=1108.752,365.986,-87.419,-178.770,14.647,150.788
C04250=1108.758,366.234,-87.455,-178.767,14.650,150.789
C04251=1108.763,366.480,-87.491,-178.765,14.653,150.789
C04252=1108.769,366.728,-87.525,-178.761,14.657,150.789
C04253=1108.775,366.975,-87.560,-178.758,14.660,150.789
C04254=1108.781,367.222,-87.596,-178.756,14.663,150.789
C04255=1108.786,367.470,-87.630,-178.752,14.667,150.789
C04256=1108.792,367.718,-87.666,-178.749,14.670,150.789
C04257=1108.797,367.965,-87.701,-178.747,14.673,150.789
C04258=1108.803,368.212,-87.737,-178.744,14.676,150.790
C04259=1108.808,368.460,-87.772,-178.740,14.679,150.790
C04260=1108.814,368.707,-87.807,-178.738,14.682,150.790
C04261=1108.820,368.955,-87.843,-178.735,14.685,150.790
C04262=1108.825,369.202,-87.878,-178.732,14.689,150.790
C04263=1108.834,369.587,-87.933,-178.728,14.694,150.791
C04264=1108.843,369.972,-87.989,-178.723,14.699,150.791
C04265=1108.852,370.356,-88.043,-178.719,14.704,150.791
C04266=1108.861,370.742,-88.098,-178.715,14.709,150.791
C04267=1108.866,370.989,-88.134,-178.711,14.712,150.792
C04268=1108.872,371.236,-88.169,-178.708,14.716,150.792
C04269=1108.878,371.483,-88.205,-178.706,14.719,150.792
C04270=1108.884,371.731,-88.241,-178.703,14.723,150.792
C04271=1108.889,371.978,-88.276,-178.700,14.726,150.792
C04272=1108.895,372.225,-88.312,-178.697,14.729,150.793
C04273=1108.900,372.473,-88.348,-178.694,14.733,150.793
C04274=1108.906,372.720,-88.383,-178.692,14.736,150.793
C04275=1108.911,372.967,-88.419,-178.689,14.739,150.793
C04276=1108.917,373.215,-88.454,-178.686,14.743,150.793
C04277=1108.923,373.462,-88.490,-178.683,14.746,150.794
C04278=1108.929,373.710,-88.526,-178.681,14.749,150.794
C04279=1108.934,373.957,-88.561,-178.677,14.753,150.794
C04280=1108.940,374.204,-88.597,-178.675,14.756,150.794
C04281=1108.946,374.451,-88.632,-178.672,14.760,150.795
C04282=1108.952,374.699,-88.668,-178.669,14.763,150.795
C04283=1108.956,374.946,-88.704,-178.667,14.766,150.795
C04284=1108.963,375.193,-88.740,-178.663,14.770,150.795
C04285=1108.968,375.440,-88.775,-178.661,14.774,150.796
C04286=1108.974,375.688,-88.811,-178.658,14.778,150.796
C04287=1108.979,375.935,-88.847,-178.655,14.781,150.796
C04288=1108.985,376.183,-88.883,-178.653,14.785,150.797
C04289=1108.991,376.430,-88.919,-178.650,14.788,150.797
C04290=1108.997,376.677,-88.955,-178.647,14.792,150.797
C04291=1109.002,376.925,-88.991,-178.644,14.796,150.798
C04292=1109.007,377.172,-89.026,-178.642,14.799,150.798
C04293=1109.014,377.419,-89.063,-178.639,14.803,150.798
C04294=1109.018,377.666,-89.099,-178.636,14.807,150.799
C04295=1109.024,377.914,-89.135,-178.633,14.810,150.799
C04296=1109.030,378.160,-89.171,-178.631,14.814,150.799
C04297=1109.035,378.408,-89.207,-178.629,14.817,150.799
C04298=1109.041,378.656,-89.243,-178.626,14.821,150.800
C04299=1109.047,378.902,-89.279,-178.623,14.825,150.800
C04300=1109.053,379.150,-89.315,-178.620,14.829,150.800
C04301=1109.058,379.397,-89.350,-178.618,14.832,150.801
C04302=1109.064,379.644,-89.387,-178.615,14.836,150.801
C04303=1109.070,379.892,-89.423,-178.612,14.840,150.802
C04304=1109.075,380.139,-89.459,-178.610,14.844,150.802
C04305=1109.081,380.386,-89.495,-178.607,14.848,150.802
C04306=1109.086,380.633,-89.532,-178.604,14.852,150.803
C04307=1109.092,380.881,-89.567,-178.602,14.855,150.803
C04308=1109.098,381.128,-89.604,-178.599,14.859,150.803
C04309=1109.103,381.375,-89.640,-178.597,14.863,150.804
C04310=1109.110,381.622,-89.676,-178.594,14.867,150.804
C04311=1109.115,381.870,-89.713,-178.592,14.871,150.805
C04312=1109.121,382.116,-89.749,-178.588,14.875,150.805
C04313=1109.126,382.364,-89.785,-178.585,14.879,150.805
C04314=1109.132,382.611,-89.821,-178.583,14.882,150.806
C04315=1109.141,383.022,-89.882,-178.579,14.890,150.807
C04316=1109.151,383.434,-89.942,-178.575,14.896,150.807
C04317=1109.160,383.846,-90.003,-178.570,14.903,150.808
C04318=1109.170,384.258,-90.064,-178.566,14.910,150.809
C04319=1109.175,384.504,-90.100,-178.564,14.913,150.809
C04320=1109.180,384.752,-90.137,-178.561,14.918,150.810
C04321=1109.187,384.999,-90.173,-178.559,14.921,150.810
C04322=1109.192,385.246,-90.210,-178.556,14.926,150.811
C04323=1109.197,385.493,-90.247,-178.553,14.930,150.811
C04324=1109.204,385.740,-90.283,-178.551,14.934,150.812
C04325=1109.208,385.988,-90.319,-178.548,14.938,150.812
C04326=1109.215,386.235,-90.356,-178.546,14.943,150.813
C04327=1109.220,386.482,-90.393,-178.543,14.946,150.813
C04328=1109.225,386.729,-90.429,-178.541,14.951,150.814
C04329=1109.232,386.976,-90.466,-178.539,14.955,150.814
C04330=1109.237,387.224,-90.502,-178.536,14.959,150.815
C04331=1109.242,387.471,-90.539,-178.533,14.964,150.815
C04332=1109.248,387.717,-90.575,-178.531,14.967,150.816
C04333=1109.254,387.965,-90.612,-178.529,14.972,150.816
C04334=1109.259,388.212,-90.649,-178.526,14.977,150.817
C04335=1109.265,388.460,-90.686,-178.524,14.980,150.817
C04336=1109.271,388.706,-90.722,-178.521,14.985,150.818
C04337=1109.276,388.953,-90.760,-178.519,14.989,150.818
C04338=1109.282,389.201,-90.797,-178.516,14.994,150.819
C04339=1109.288,389.448,-90.834,-178.514,14.998,150.820
C04340=1109.293,389.694,-90.870,-178.511,15.003,150.820
C04341=1109.299,389.942,-90.907,-178.509,15.007,150.821
C04342=1109.304,390.189,-90.944,-178.507,15.011,150.821
C04343=1109.310,390.436,-90.981,-178.504,15.015,150.822
C04344=1109.316,390.683,-91.017,-178.501,15.020,150.822
C04345=1109.322,390.929,-91.055,-178.499,15.025,150.823
C04346=1109.327,391.177,-91.092,-178.497,15.029,150.824
C04347=1109.333,391.424,-91.129,-178.495,15.033,150.824
C04348=1109.338,391.672,-91.166,-178.492,15.038,150.825
C04349=1109.345,391.919,-91.202,-178.490,15.042,150.825
C04350=1109.350,392.166,-91.239,-178.487,15.047,150.826
C04351=1109.356,392.413,-91.276,-178.485,15.051,150.827
C04352=1109.362,392.660,-91.314,-178.483,15.056,150.827
C04353=1109.367,392.907,-91.351,-178.481,15.060,150.828
C04354=1109.373,393.154,-91.388,-178.478,15.065,150.829
C04355=1109.378,393.402,-91.425,-178.476,15.070,150.829
C04356=1109.384,393.649,-91.462,-178.473,15.074,150.830
C04357=1109.390,393.896,-91.500,-178.471,15.079,150.831
C04358=1109.395,394.143,-91.537,-178.469,15.083,150.831
C04359=1109.401,394.390,-91.574,-178.467,15.088,150.832
C04360=1109.407,394.637,-91.611,-178.464,15.093,150.833
C04361=1109.412,394.884,-91.648,-178.462,15.098,150.833
C04362=1109.417,395.131,-91.685,-178.460,15.103,150.834
C04363=1109.423,395.378,-91.722,-178.458,15.107,150.835
C04364=1109.429,395.625,-91.760,-178.455,15.112,150.835
C04365=1109.434,395.873,-91.797,-178.453,15.117,150.836
C04366=1109.440,396.119,-91.835,-178.451,15.122,150.837
C04367=1109.445,396.331,-91.866,-178.449,15.126,150.838
C04368=1109.451,396.543,-91.898,-178.447,15.130,150.838
C04369=1109.455,396.755,-91.930,-178.445,15.134,150.839
C04370=1109.460,396.966,-91.962,-178.443,15.139,150.840
C04371=1109.464,397.179,-91.995,-178.441,15.143,150.840
C04372=1109.469,397.390,-92.027,-178.440,15.147,150.841
C04373=1109.475,397.602,-92.058,-178.438,15.151,150.841
C04374=1109.479,397.814,-92.091,-178.436,15.155,150.842
C04375=1109.484,398.061,-92.128,-178.434,15.160,150.843
C04376=1109.490,398.308,-92.166,-178.431,15.165,150.844
C04377=1109.496,398.555,-92.203,-178.429,15.170,150.844
C04378=1109.502,398.802,-92.241,-178.427,15.175,150.845
C04379=1109.507,399.050,-92.278,-178.425,15.180,150.846
C04380=1109.513,399.296,-92.316,-178.423,15.185,150.847
C04381=1109.518,399.543,-92.354,-178.420,15.190,150.848
C04382=1109.524,399.790,-92.391,-178.418,15.196,150.849
C04383=1109.530,400.037,-92.429,-178.416,15.201,150.849
C04384=1109.535,400.285,-92.466,-178.414,15.206,150.850
C04385=1109.541,400.532,-92.504,-178.412,15.210,150.851
C04386=1109.547,400.778,-92.542,-178.410,15.216,150.852
C04387=1109.552,401.026,-92.579,-178.408,15.221,150.853
C04388=1109.557,401.273,-92.617,-178.406,15.226,150.854
C04389=1109.563,401.520,-92.655,-178.404,15.231,150.855
C04390=1109.568,401.767,-92.692,-178.402,15.237,150.855
C04391=1109.574,402.014,-92.730,-178.400,15.242,150.856
C04392=1109.580,402.261,-92.768,-178.398,15.247,150.857
C04393=1109.585,402.508,-92.806,-178.396,15.252,150.858
C04394=1109.591,402.755,-92.843,-178.393,15.258,150.859
C04395=1109.597,403.003,-92.881,-178.391,15.264,150.860
C04396=1109.602,403.250,-92.920,-178.389,15.269,150.861
C04397=1109.608,403.496,-92.958,-178.387,15.274,150.862
C04398=1109.614,403.744,-92.995,-178.385,15.280,150.863
C04399=1109.619,403.991,-93.033,-178.383,15.285,150.864
C04400=1109.625,404.238,-93.071,-178.381,15.290,150.865
C04401=1109.630,404.485,-93.109,-178.379,15.296,150.865
C04402=1109.636,404.731,-93.147,-178.377,15.301,150.866
C04403=1109.643,404.979,-93.185,-178.375,15.306,150.867
C04404=1109.648,405.226,-93.223,-178.374,15.312,150.868
C04405=1109.654,405.473,-93.261,-178.372,15.318,150.869
C04406=1109.659,405.720,-93.299,-178.369,15.324,150.870
C04407=1109.664,405.967,-93.336,-178.367,15.329,150.871
C04408=1109.670,406.214,-93.375,-178.365,15.335,150.872
C04409=1109.675,406.461,-93.413,-178.363,15.340,150.873
C04410=1109.681,406.708,-93.451,-178.361,15.346,150.874
C04411=1109.687,406.955,-93.489,-178.360,15.351,150.875
C04412=1109.692,407.202,-93.527,-178.358,15.357,150.876
C04413=1109.698,407.449,-93.566,-178.355,15.363,150.877
C04414=1109.704,407.696,-93.604,-178.354,15.369,150.878
C04415=1109.709,407.943,-93.643,-178.352,15.375,150.880
C04416=1109.715,408.189,-93.680,-178.350,15.380,150.881
C04417=1109.721,408.437,-93.719,-178.348,15.387,150.882
C04418=1109.726,408.684,-93.757,-178.346,15.392,150.883
C04419=1109.732,408.931,-93.795,-178.344,15.398,150.884
C04420=1109.737,409.178,-93.833,-178.343,15.404,150.885
C04421=1109.742,409.425,-93.872,-178.340,15.410,150.886
C04422=1109.749,409.672,-93.911,-178.339,15.416,150.887
C04423=1109.753,409.883,-93.943,-178.337,15.420,150.888
C04424=1109.757,410.095,-93.976,-178.336,15.426,150.889
C04425=1109.762,410.307,-94.009,-178.334,15.431,150.890
C04426=1109.767,410.518,-94.042,-178.332,15.436,150.891
C04427=1109.772,410.729,-94.075,-178.331,15.442,150.892
C04428=1109.777,410.941,-94.107,-178.329,15.446,150.893
C04429=1109.782,411.152,-94.141,-178.328,15.452,150.894
C04430=1109.786,411.364,-94.174,-178.326,15.457,150.895
C04431=1109.791,411.611,-94.212,-178.324,15.464,150.896
C04432=1109.798,411.858,-94.251,-178.323,15.469,150.897
C04433=1109.803,412.105,-94.289,-178.321,15.475,150.899
C04434=1109.808,412.352,-94.328,-178.319,15.482,150.900
C04435=1109.814,412.598,-94.367,-178.317,15.488,150.901
C04436=1109.820,412.846,-94.405,-178.316,15.493,150.902
C04437=1109.826,413.093,-94.443,-178.314,15.500,150.903
C04438=1109.831,413.339,-94.482,-178.312,15.506,150.905
C04439=1109.836,413.586,-94.520,-178.310,15.513,150.906
C04440=1109.842,413.833,-94.560,-178.309,15.519,150.907
C04441=1109.847,414.080,-94.598,-178.307,15.525,150.908
C04442=1109.854,414.326,-94.637,-178.305,15.532,150.909
C04443=1109.859,414.574,-94.675,-178.303,15.538,150.911
C04444=1109.865,414.821,-94.715,-178.301,15.544,150.912
C04445=1109.870,415.068,-94.753,-178.300,15.551,150.913
C04446=1109.876,415.315,-94.792,-178.298,15.558,150.915
C04447=1109.881,415.562,-94.831,-178.297,15.564,150.916
C04448=1109.888,415.808,-94.869,-178.295,15.570,150.917
C04449=1109.893,416.056,-94.908,-178.293,15.576,150.918
C04450=1109.899,416.302,-94.947,-178.291,15.583,150.920
C04451=1109.904,416.549,-94.986,-178.290,15.590,150.921
C04452=1109.910,416.796,-95.025,-178.288,15.596,150.922
C04453=1109.915,417.043,-95.064,-178.287,15.603,150.924
C04454=1109.921,417.289,-95.103,-178.285,15.610,150.925
C04455=1109.927,417.537,-95.142,-178.283,15.616,150.926
C04456=1109.932,417.783,-95.181,-178.282,15.623,150.928
C04457=1109.938,418.030,-95.220,-178.281,15.629,150.929
C04458=1109.943,418.278,-95.258,-178.279,15.637,150.931
C04459=1109.949,418.524,-95.297,-178.277,15.643,150.932
C04460=1109.955,418.771,-95.337,-178.275,15.650,150.933
C04461=1109.960,419.018,-95.376,-178.274,15.657,150.935
C04462=1109.966,419.265,-95.414,-178.273,15.663,150.936
C04463=1109.971,419.512,-95.454,-178.271,15.670,150.938
C04464=1109.976,419.759,-95.493,-178.269,15.678,150.939
C04465=1109.982,420.005,-95.532,-178.268,15.684,150.941
C04466=1109.988,420.252,-95.572,-178.266,15.691,150.942
C04467=1109.993,420.499,-95.611,-178.264,15.698,150.943
C04468=1109.999,420.746,-95.650,-178.264,15.705,150.945
C04469=1110.005,420.993,-95.689,-178.262,15.712,150.946
C04470=1110.010,421.239,-95.728,-178.260,15.719,150.948
C04471=1110.016,421.486,-95.767,-178.259,15.726,150.949
C04472=1110.021,421.733,-95.807,-178.257,15.733,150.951
C04473=1110.027,421.980,-95.846,-178.256,15.741,150.952
C04474=1110.033,422.227,-95.885,-178.255,15.748,150.954
C04475=1110.039,422.474,-95.925,-178.253,15.755,150.955
C04476=1110.044,422.720,-95.964,-178.251,15.762,150.957
C04477=1110.050,422.967,-96.003,-178.250,15.770,150.959
C04478=1110.055,423.214,-96.043,-178.249,15.776,150.960
C04479=1110.061,423.432,-96.078,-178.247,15.783,150.961
C04480=1110.065,423.649,-96.112,-178.246,15.790,150.963
C04481=1110.070,423.867,-96.147,-178.245,15.796,150.964
C04482=1110.075,424.085,-96.182,-178.244,15.803,150.966
C04483=1110.080,424.303,-96.217,-178.243,15.809,150.967
C04484=1110.084,424.520,-96.252,-178.242,15.815,150.968
C04485=1110.089,424.739,-96.287,-178.240,15.822,150.970
C04486=1110.094,424.957,-96.322,-178.240,15.829,150.971
C04487=1110.100,425.204,-96.361,-178.238,15.836,150.973
C04488=1110.105,425.450,-96.402,-178.237,15.844,150.975
C04489=1110.111,425.696,-96.441,-178.235,15.851,150.976
C04490=1110.117,425.943,-96.480,-178.234,15.859,150.978
C04491=1110.121,426.190,-96.520,-178.232,15.867,150.980
C04492=1110.128,426.437,-96.559,-178.232,15.874,150.981
C04493=1110.133,426.683,-96.599,-178.231,15.882,150.983
C04494=1110.139,426.931,-96.639,-178.229,15.889,150.985
C04495=1110.144,427.177,-96.678,-178.228,15.897,150.987
C04496=1110.150,427.424,-96.719,-178.227,15.905,150.988
C04497=1110.155,427.670,-96.758,-178.226,15.913,150.990
C04498=1110.161,427.917,-96.797,-178.224,15.921,150.992
C04499=1110.166,428.164,-96.838,-178.223,15.929,150.994
C04500=1110.172,428.411,-96.877,-178.222,15.936,150.995
C04501=1110.178,428.658,-96.918,-178.220,15.944,150.997
C04502=1110.184,428.904,-96.957,-178.219,15.952,150.999
C04503=1110.189,429.151,-96.998,-178.218,15.960,151.001
C04504=1110.195,429.397,-97.037,-178.217,15.968,151.002
C04505=1110.200,429.645,-97.077,-178.216,15.976,151.004
C04506=1110.206,429.890,-97.116,-178.215,15.984,151.006
C04507=1110.211,430.138,-97.156,-178.214,15.992,151.008
C04508=1110.217,430.384,-97.196,-178.213,16.000,151.010
C04509=1110.223,430.631,-97.237,-178.212,16.009,151.012
C04510=1110.228,430.877,-97.276,-178.211,16.017,151.014
C04511=1110.234,431.124,-97.317,-178.210,16.025,151.016
C04512=1110.238,431.371,-97.356,-178.209,16.033,151.017
C04513=1110.245,431.617,-97.397,-178.208,16.041,151.019
C04514=1110.250,431.865,-97.437,-178.207,16.049,151.021
C04515=1110.256,432.110,-97.476,-178.206,16.058,151.023
C04516=1110.262,432.357,-97.517,-178.205,16.066,151.025
C04517=1110.266,432.604,-97.557,-178.204,16.074,151.027
C04518=1110.273,432.850,-97.597,-178.203,16.083,151.029
C04519=1110.278,433.097,-97.637,-178.202,16.091,151.031
C04520=1110.283,433.343,-97.678,-178.202,16.100,151.033
C04521=1110.289,433.590,-97.718,-178.201,16.108,151.035
C04522=1110.294,433.837,-97.758,-178.199,16.117,151.037
C04523=1110.300,434.083,-97.799,-178.198,16.126,151.039
C04524=1110.306,434.329,-97.838,-178.198,16.134,151.041
C04525=1110.311,434.577,-97.878,-178.197,16.143,151.043
C04526=1110.317,434.824,-97.919,-178.196,16.151,151.045
C04527=1110.322,435.070,-97.960,-178.196,16.160,151.047
C04528=1110.328,435.316,-98.000,-178.194,16.169,151.049
C04529=1110.333,435.562,-98.040,-178.194,16.178,151.052
C04530=1110.339,435.809,-98.081,-178.193,16.187,151.054
C04531=1110.345,436.056,-98.122,-178.193,16.195,151.056
C04532=1110.349,436.303,-98.161,-178.192,16.204,151.058
C04533=1110.355,436.549,-98.202,-178.191,16.213,151.060
C04534=1110.360,436.796,-98.242,-178.190,16.222,151.062
C04535=1110.366,437.028,-98.280,-178.189,16.231,151.064
C04536=1110.371,437.261,-98.319,-178.189,16.239,151.066
C04537=1110.377,437.492,-98.357,-178.189,16.247,151.068
C04538=1110.382,437.725,-98.396,-178.188,16.256,151.070
C04539=1110.387,437.958,-98.434,-178.187,16.265,151.073
C04540=1110.392,438.190,-98.472,-178.187,16.273,151.075
C04541=1110.397,438.423,-98.511,-178.186,16.282,151.077
C04542=1110.403,438.656,-98.549,-178.186,16.290,151.079
C04543=1110.408,438.902,-98.589,-178.185,16.299,151.081
C04544=1110.413,439.149,-98.630,-178.184,16.309,151.083
C04545=1110.419,439.396,-98.671,-178.184,16.318,151.086
C04546=1110.425,439.642,-98.711,-178.184,16.327,151.088
C04547=1110.430,439.889,-98.752,-178.183,16.337,151.090
C04548=1110.436,440.135,-98.793,-178.182,16.346,151.093
C04549=1110.441,440.382,-98.834,-178.182,16.356,151.095
C04550=1110.447,440.628,-98.875,-178.181,16.365,151.097
C04551=1110.452,440.875,-98.915,-178.181,16.375,151.100
C04552=1110.458,441.121,-98.956,-178.181,16.384,151.102
C04553=1110.464,441.368,-98.997,-178.180,16.394,151.104
C04554=1110.469,441.614,-99.038,-178.180,16.403,151.107
C04555=1110.474,441.861,-99.078,-178.179,16.413,151.109
C04556=1110.480,442.107,-99.120,-178.179,16.423,151.112
C04557=1110.485,442.353,-99.160,-178.179,16.432,151.114
C04558=1110.491,442.600,-99.201,-178.178,16.443,151.117
C04559=1110.497,442.846,-99.242,-178.178,16.452,151.119
C04560=1110.503,443.093,-99.283,-178.178,16.462,151.122
C04561=1110.508,443.338,-99.324,-178.178,16.472,151.124
C04562=1110.513,443.585,-99.365,-178.178,16.482,151.127
C04563=1110.518,443.832,-99.406,-178.177,16.492,151.129
C04564=1110.524,444.078,-99.447,-178.177,16.502,151.132
C04565=1110.529,444.325,-99.488,-178.177,16.512,151.134
C04566=1110.535,444.571,-99.530,-178.178,16.522,151.137
C04567=1110.540,444.818,-99.571,-178.178,16.532,151.140
C04568=1110.546,445.064,-99.612,-178.179,16.540,151.142
C04569=1110.551,445.310,-99.653,-178.180,16.551,151.145
C04570=1110.557,445.556,-99.694,-178.180,16.561,151.148
C04571=1110.563,445.803,-99.735,-178.181,16.570,151.150
C04572=1110.568,446.050,-99.777,-178.182,16.580,151.153
C04573=1110.574,446.297,-99.818,-178.183,16.590,151.156
C04574=1110.580,446.543,-99.859,-178.184,16.599,151.158
C04575=1110.584,446.789,-99.900,-178.186,16.609,151.161
C04576=1110.590,447.035,-99.942,-178.187,16.619,151.164
C04577=1110.596,447.282,-99.982,-178.188,16.628,151.167
C04578=1110.601,447.529,-100.024,-178.190,16.638,151.170
C04579=1110.606,447.776,-100.065,-178.191,16.648,151.172
C04580=1110.612,448.021,-100.106,-178.193,16.658,151.175
C04581=1110.617,448.268,-100.148,-178.195,16.667,151.178
C04582=1110.623,448.514,-100.189,-178.196,16.677,151.181
C04583=1110.628,448.761,-100.231,-178.198,16.686,151.184
C04584=1110.633,449.008,-100.272,-178.200,16.696,151.187
C04585=1110.639,449.254,-100.313,-178.202,16.705,151.190
C04586=1110.645,449.500,-100.355,-178.205,16.714,151.192
C04587=1110.650,449.747,-100.396,-178.206,16.725,151.195
C04588=1110.656,449.993,-100.437,-178.209,16.734,151.198
C04589=1110.661,450.239,-100.479,-178.211,16.743,151.201
C04590=1110.666,450.486,-100.520,-178.214,16.753,151.204
C04591=1110.255,450.480,-100.622,-178.302,16.987,151.283
C04592=1110.250,450.233,-100.581,-178.299,16.977,151.280
C04593=1110.245,449.988,-100.540,-178.297,16.968,151.277
C04594=1110.239,449.742,-100.498,-178.295,16.958,151.274
C04595=1110.234,449.495,-100.456,-178.293,16.948,151.271
C04596=1110.228,449.248,-100.415,-178.291,16.939,151.268
C04597=1110.223,449.002,-100.373,-178.289,16.929,151.265
C04598=1110.217,448.756,-100.332,-178.287,16.919,151.262
C04599=1110.211,448.509,-100.291,-178.285,16.910,151.259
C04600=1110.206,448.262,-100.249,-178.283,16.900,151.256
C04601=1110.200,448.016,-100.208,-178.282,16.890,151.253
C04602=1110.196,447.770,-100.167,-178.280,16.881,151.251
C04603=1110.190,447.523,-100.125,-178.278,16.871,151.248
C04604=1110.184,447.277,-100.084,-178.277,16.861,151.245
C04605=1110.179,447.030,-100.042,-178.275,16.851,151.242
C04606=1110.173,446.784,-100.001,-178.274,16.841,151.239
C04607=1110.168,446.537,-99.960,-178.273,16.832,151.237
C04608=1110.163,446.291,-99.918,-178.272,16.821,151.234
C04609=1110.157,446.045,-99.877,-178.271,16.812,151.231
C04610=1110.151,445.798,-99.836,-178.270,16.802,151.228
C04611=1110.146,445.552,-99.794,-178.269,16.792,151.226
C04612=1110.140,445.305,-99.753,-178.268,16.782,151.223
C04613=1110.134,445.059,-99.712,-178.268,16.773,151.220
C04614=1110.129,444.813,-99.672,-178.268,16.763,151.218
C04615=1110.124,444.566,-99.630,-178.267,16.753,151.215
C04616=1110.119,444.319,-99.589,-178.267,16.743,151.212
C04617=1110.113,444.073,-99.547,-178.267,16.733,151.210
C04618=1110.107,443.826,-99.507,-178.267,16.723,151.207
C04619=1110.102,443.580,-99.465,-178.267,16.713,151.205
C04620=1110.097,443.334,-99.424,-178.266,16.703,151.202
C04621=1110.091,443.087,-99.383,-178.267,16.693,151.200
C04622=1110.085,442.841,-99.342,-178.267,16.683,151.197
C04623=1110.080,442.595,-99.301,-178.268,16.673,151.195
C04624=1110.074,442.348,-99.260,-178.268,16.663,151.192
C04625=1110.068,442.101,-99.219,-178.269,16.653,151.190
C04626=1110.063,441.855,-99.178,-178.269,16.644,151.187
C04627=1110.058,441.609,-99.137,-178.270,16.633,151.185
C04628=1110.053,441.362,-99.096,-178.270,16.624,151.182
C04629=1110.047,441.116,-99.055,-178.270,16.615,151.180
C04630=1110.041,440.869,-99.014,-178.271,16.604,151.177
C04631=1110.036,440.623,-98.974,-178.271,16.595,151.175
C04632=1110.030,440.377,-98.932,-178.272,16.585,151.173
C04633=1110.024,440.130,-98.891,-178.272,16.576,151.170
C04634=1110.019,439.884,-98.851,-178.272,16.567,151.168
C04635=1110.014,439.637,-98.810,-178.273,16.557,151.166
C04636=1110.008,439.390,-98.770,-178.274,16.547,151.163
C04637=1110.002,439.144,-98.728,-178.274,16.539,151.161
C04638=1109.996,438.898,-98.688,-178.275,16.529,151.159
C04639=1109.991,438.651,-98.648,-178.276,16.519,151.157
C04640=1109.985,438.420,-98.609,-178.276,16.511,151.155
C04641=1109.980,438.188,-98.571,-178.277,16.502,151.152
C04642=1109.975,437.956,-98.533,-178.278,16.493,151.150
C04643=1109.970,437.724,-98.495,-178.278,16.485,151.148
C04644=1109.965,437.493,-98.457,-178.279,16.476,151.146
C04645=1109.959,437.261,-98.419,-178.280,16.467,151.144
C04646=1109.954,437.030,-98.380,-178.280,16.459,151.142
C04647=1109.949,436.798,-98.343,-178.281,16.451,151.140
C04648=1109.943,436.551,-98.302,-178.282,16.441,151.138
C04649=1109.938,436.304,-98.261,-178.282,16.432,151.136
C04650=1109.933,436.058,-98.221,-178.283,16.423,151.133
C04651=1109.927,435.811,-98.180,-178.284,16.415,151.131
C04652=1109.922,435.565,-98.140,-178.285,16.405,151.129
C04653=1109.916,435.318,-98.099,-178.285,16.396,151.127
C04654=1109.910,435.072,-98.059,-178.286,16.388,151.125
C04655=1109.905,434.825,-98.018,-178.287,16.379,151.123
C04656=1109.899,434.579,-97.978,-178.288,16.371,151.121
C04657=1109.894,434.333,-97.937,-178.289,16.361,151.119
C04658=1109.888,434.085,-97.898,-178.290,16.353,151.117
C04659=1109.883,433.839,-97.857,-178.291,16.344,151.115
C04660=1109.878,433.592,-97.817,-178.291,16.335,151.112
C04661=1109.872,433.346,-97.776,-178.292,16.327,151.111
C04662=1109.866,433.100,-97.736,-178.293,16.319,151.109
C04663=1109.861,432.852,-97.696,-178.295,16.309,151.106
C04664=1109.855,432.606,-97.655,-178.295,16.301,151.104
C04665=1109.849,432.360,-97.616,-178.296,16.293,151.103
C04666=1109.844,432.112,-97.576,-178.297,16.284,151.101
C04667=1109.839,431.866,-97.535,-178.298,16.276,151.099
C04668=1109.833,431.620,-97.495,-178.299,16.268,151.097
C04669=1109.827,431.372,-97.455,-178.300,16.259,151.095
C04670=1109.822,431.126,-97.415,-178.301,16.251,151.093
C04671=1109.816,430.880,-97.374,-178.302,16.243,151.091
C04672=1109.811,430.633,-97.335,-178.303,16.234,151.089
C04673=1109.805,430.386,-97.295,-178.304,16.226,151.087
C04674=1109.800,430.140,-97.254,-178.305,16.218,151.085
C04675=1109.794,429.893,-97.215,-178.306,16.210,151.083
C04676=1109.789,429.647,-97.174,-178.308,16.202,151.082
C04677=1109.783,429.399,-97.134,-178.309,16.194,151.080
C04678=1109.777,429.153,-97.094,-178.310,16.186,151.078
C04679=1109.771,428.907,-97.055,-178.311,16.178,151.076
C04680=1109.766,428.660,-97.014,-178.312,16.170,151.074
C04681=1109.760,428.413,-96.975,-178.313,16.162,151.073
C04682=1109.755,428.166,-96.935,-178.315,16.154,151.071
C04683=1109.749,427.920,-96.896,-178.316,16.146,151.069
C04684=1109.744,427.673,-96.856,-178.317,16.138,151.067
C04685=1109.738,427.427,-96.816,-178.318,16.130,151.065
C04686=1109.732,427.180,-96.776,-178.320,16.122,151.064
C04687=1109.727,426.932,-96.736,-178.321,16.114,151.062
C04688=1109.721,426.686,-96.697,-178.322,16.107,151.060
C04689=1109.716,426.439,-96.657,-178.324,16.099,151.058
C04690=1109.710,426.192,-96.617,-178.325,16.091,151.057
C04691=1109.704,425.946,-96.577,-178.326,16.083,151.055
C04692=1109.699,425.699,-96.538,-178.328,16.076,151.053
C04693=1109.693,425.452,-96.498,-178.328,16.069,151.052
C04694=1109.688,425.205,-96.459,-178.330,16.061,151.050
C04695=1109.682,424.960,-96.419,-178.331,16.053,151.048
C04696=1109.678,424.741,-96.384,-178.332,16.047,151.047
C04697=1109.673,424.523,-96.349,-178.334,16.040,151.046
C04698=1109.668,424.305,-96.314,-178.335,16.033,151.044
C04699=1109.663,424.087,-96.279,-178.336,16.026,151.043
C04700=1109.658,423.869,-96.244,-178.338,16.020,151.041
C04701=1109.653,423.651,-96.209,-178.338,16.013,151.040
C04702=1109.648,423.433,-96.174,-178.340,16.007,151.038
C04703=1109.644,423.215,-96.140,-178.341,16.000,151.037
C04704=1109.637,422.969,-96.100,-178.342,15.993,151.035
C04705=1109.632,422.722,-96.061,-178.344,15.985,151.034
C04706=1109.626,422.475,-96.021,-178.346,15.978,151.032
C04707=1109.620,422.229,-95.982,-178.347,15.971,151.031
C04708=1109.615,421.981,-95.942,-178.348,15.964,151.029
C04709=1109.609,421.735,-95.903,-178.350,15.956,151.028
C04710=1109.603,421.488,-95.864,-178.352,15.949,151.026
C04711=1109.598,421.241,-95.825,-178.353,15.942,151.025
C04712=1109.592,420.995,-95.785,-178.354,15.935,151.023
C04713=1109.586,420.748,-95.746,-178.356,15.928,151.022
C04714=1109.582,420.501,-95.706,-178.357,15.921,151.020
C04715=1109.576,420.253,-95.668,-178.359,15.914,151.019
C04716=1109.570,420.007,-95.629,-178.360,15.907,151.017
C04717=1109.564,419.760,-95.589,-178.362,15.900,151.016
C04718=1109.559,419.513,-95.550,-178.364,15.893,151.014
C04719=1109.553,419.267,-95.511,-178.365,15.886,151.013
C04720=1109.547,419.020,-95.472,-178.366,15.879,151.011
C04721=1109.542,418.773,-95.433,-178.368,15.872,151.010
C04722=1109.537,418.526,-95.394,-178.370,15.865,151.008
C04723=1109.531,418.279,-95.355,-178.371,15.859,151.007
C04724=1109.525,418.033,-95.316,-178.373,15.852,151.006
C04725=1109.520,417.785,-95.276,-178.375,15.844,151.004
C04726=1109.515,417.538,-95.237,-178.376,15.838,151.003
C04727=1109.509,417.292,-95.198,-178.378,15.831,151.001
C04728=1109.503,417.045,-95.159,-178.379,15.825,151.000
C04729=1109.498,416.797,-95.120,-178.381,15.817,150.999
C04730=1109.492,416.551,-95.081,-178.383,15.811,150.997
C04731=1109.486,416.304,-95.043,-178.384,15.804,150.996
C04732=1109.480,416.057,-95.004,-178.387,15.798,150.995
C04733=1109.475,415.811,-94.965,-178.388,15.791,150.993
C04734=1109.469,415.564,-94.926,-178.390,15.784,150.992
C04735=1109.464,415.317,-94.887,-178.391,15.778,150.991
C04736=1109.458,415.070,-94.848,-178.393,15.771,150.989
C04737=1109.452,414.822,-94.810,-178.395,15.765,150.988
C04738=1109.447,414.576,-94.771,-178.397,15.758,150.987
C04739=1109.441,414.329,-94.733,-178.398,15.752,150.986
C04740=1109.435,414.082,-94.693,-178.400,15.746,150.985
C04741=1109.430,413.835,-94.655,-178.402,15.739,150.983
C04742=1109.424,413.589,-94.616,-178.403,15.733,150.982
C04743=1109.419,413.341,-94.577,-178.405,15.727,150.981
C04744=1109.413,413.094,-94.538,-178.407,15.720,150.979
C04745=1109.407,412.848,-94.500,-178.409,15.714,150.978
C04746=1109.401,412.600,-94.461,-178.411,15.708,150.977
C04747=1109.396,412.353,-94.423,-178.412,15.702,150.976
C04748=1109.391,412.106,-94.384,-178.414,15.695,150.975
C04749=1109.385,411.860,-94.346,-178.416,15.689,150.973
C04750=1109.379,411.612,-94.307,-178.418,15.683,150.972
C04751=1109.374,411.365,-94.269,-178.420,15.677,150.971
C04752=1109.369,411.155,-94.235,-178.421,15.671,150.970
C04753=1109.364,410.943,-94.202,-178.423,15.666,150.969
C04754=1109.359,410.730,-94.169,-178.425,15.661,150.968
C04755=1109.355,410.520,-94.136,-178.426,15.656,150.967
C04756=1109.349,410.308,-94.104,-178.428,15.650,150.966
C04757=1109.345,410.096,-94.071,-178.429,15.646,150.965
C04758=1109.340,409.884,-94.038,-178.431,15.640,150.964
C04759=1109.335,409.673,-94.005,-178.433,15.635,150.963
C04760=1109.330,409.426,-93.966,-178.434,15.629,150.962
C04761=1109.324,409.179,-93.928,-178.436,15.623,150.961
C04762=1109.319,408.932,-93.890,-178.438,15.617,150.960
C04763=1109.313,408.685,-93.851,-178.440,15.611,150.959
C04764=1109.307,408.438,-93.814,-178.442,15.605,150.957
C04765=1109.302,408.192,-93.775,-178.443,15.599,150.956
C04766=1109.297,407.945,-93.736,-178.446,15.593,150.955
C04767=1109.290,407.697,-93.698,-178.448,15.587,150.954
C04768=1109.285,407.450,-93.660,-178.449,15.582,150.953
C04769=1109.279,407.203,-93.622,-178.451,15.576,150.952
C04770=1109.274,406.956,-93.584,-178.453,15.571,150.951
C04771=1109.269,406.709,-93.545,-178.455,15.564,150.950
C04772=1109.263,406.463,-93.508,-178.457,15.558,150.949
C04773=1109.257,406.215,-93.469,-178.459,15.553,150.948
C04774=1109.251,405.968,-93.431,-178.461,15.547,150.947
C04775=1109.246,405.721,-93.393,-178.463,15.542,150.946
C04776=1109.240,405.474,-93.355,-178.466,15.536,150.945
C04777=1109.235,405.227,-93.317,-178.467,15.530,150.944
C04778=1109.229,404.980,-93.279,-178.469,15.525,150.943
C04779=1109.223,404.733,-93.240,-178.471,15.519,150.942
C04780=1109.218,404.486,-93.202,-178.473,15.514,150.941
C04781=1109.212,404.239,-93.165,-178.475,15.508,150.940
C04782=1109.207,403.992,-93.127,-178.477,15.503,150.939
C04783=1109.201,403.745,-93.089,-178.479,15.497,150.938
C04784=1109.196,403.498,-93.051,-178.482,15.491,150.937
C04785=1109.190,403.251,-93.013,-178.484,15.486,150.936
C04786=1109.184,403.004,-92.975,-178.486,15.481,150.935
C04787=1109.178,402.756,-92.937,-178.487,15.475,150.934
C04788=1109.173,402.509,-92.900,-178.489,15.470,150.933
C04789=1109.167,402.262,-92.862,-178.491,15.464,150.933
C04790=1109.161,402.015,-92.824,-178.494,15.459,150.932
C04791=1109.156,401.769,-92.786,-178.496,15.454,150.931
C04792=1109.151,401.521,-92.748,-178.498,15.449,150.930
C04793=1109.145,401.274,-92.710,-178.500,15.443,150.929
C04794=1109.139,401.027,-92.673,-178.502,15.438,150.928
C04795=1109.133,400.780,-92.636,-178.504,15.433,150.927
C04796=1109.128,400.533,-92.597,-178.506,15.427,150.926
C04797=1109.122,400.286,-92.560,-178.508,15.422,150.926
C04798=1109.117,400.039,-92.523,-178.510,15.417,150.925
C04799=1109.111,399.792,-92.484,-178.512,15.412,150.924
C04800=1109.106,399.545,-92.446,-178.515,15.407,150.923
C04801=1109.100,399.298,-92.409,-178.517,15.401,150.922
C04802=1109.094,399.051,-92.372,-178.519,15.397,150.921
C04803=1109.088,398.804,-92.335,-178.521,15.391,150.920
C04804=1109.083,398.557,-92.296,-178.524,15.386,150.920
C04805=1109.078,398.309,-92.259,-178.526,15.381,150.919
C04806=1109.072,398.062,-92.221,-178.528,15.376,150.918
C04807=1109.066,397.815,-92.184,-178.530,15.371,150.917
C04808=1109.061,397.603,-92.151,-178.532,15.367,150.917
C04809=1109.056,397.392,-92.119,-178.533,15.362,150.916
C04810=1109.051,397.179,-92.088,-178.535,15.359,150.915
C04811=1109.047,396.968,-92.055,-178.537,15.354,150.915
C04812=1109.042,396.756,-92.024,-178.540,15.350,150.914
C04813=1109.037,396.544,-91.991,-178.541,15.345,150.913
C04814=1109.032,396.332,-91.959,-178.543,15.342,150.913
C04815=1109.027,396.121,-91.927,-178.545,15.337,150.912
C04816=1109.021,395.873,-91.890,-178.547,15.332,150.911
C04817=1109.017,395.626,-91.853,-178.550,15.327,150.910
C04818=1109.011,395.380,-91.815,-178.552,15.322,150.910
C04819=1109.005,395.132,-91.778,-178.554,15.317,150.909
C04820=1109.000,394.885,-91.741,-178.556,15.313,150.908
C04821=1108.994,394.638,-91.703,-178.558,15.309,150.908
C04822=1108.988,394.391,-91.666,-178.561,15.304,150.907
C04823=1108.983,394.143,-91.629,-178.563,15.299,150.906
C04824=1108.977,393.897,-91.591,-178.565,15.294,150.905
C04825=1108.971,393.649,-91.554,-178.568,15.289,150.905
C04826=1108.966,393.402,-91.517,-178.570,15.285,150.904
C04827=1108.959,393.155,-91.481,-178.572,15.280,150.903
C04828=1108.954,392.909,-91.443,-178.575,15.275,150.903
C04829=1108.948,392.661,-91.406,-178.577,15.270,150.902
C04830=1108.943,392.414,-91.369,-178.580,15.266,150.901
C04831=1108.937,392.167,-91.332,-178.581,15.261,150.901
C04832=1108.932,391.919,-91.295,-178.584,15.257,150.900
C04833=1108.926,391.673,-91.257,-178.587,15.252,150.900
C04834=1108.920,391.425,-91.220,-178.589,15.247,150.899
C04835=1108.914,391.178,-91.184,-178.591,15.243,150.898
C04836=1108.909,390.931,-91.147,-178.593,15.239,150.898
C04837=1108.903,390.684,-91.110,-178.596,15.234,150.897
C04838=1108.898,390.437,-91.073,-178.598,15.229,150.896
C04839=1108.892,390.189,-91.036,-178.600,15.225,150.896
C04840=1108.886,389.942,-91.000,-178.603,15.221,150.895
C04841=1108.880,389.696,-90.962,-178.606,15.216,150.895
C04842=1108.875,389.449,-90.925,-178.608,15.211,150.894
C04843=1108.869,389.202,-90.888,-178.610,15.207,150.893
C04844=1108.863,388.955,-90.852,-178.613,15.203,150.893
C04845=1108.857,388.707,-90.815,-178.616,15.198,150.892
C04846=1108.852,388.460,-90.778,-178.618,15.194,150.892
C04847=1108.846,388.213,-90.742,-178.620,15.190,150.891
C04848=1108.840,387.966,-90.705,-178.623,15.185,150.891
C04849=1108.835,387.718,-90.668,-178.626,15.181,150.890
C04850=1108.830,387.471,-90.632,-178.628,15.177,150.890
C04851=1108.824,387.224,-90.595,-178.630,15.172,150.889
C04852=1108.818,386.977,-90.558,-178.633,15.168,150.888
C04853=1108.812,386.730,-90.521,-178.636,15.164,150.888
C04854=1108.807,386.483,-90.485,-178.638,15.160,150.887
C04855=1108.801,386.236,-90.448,-178.640,15.155,150.887
C04856=1108.796,385.989,-90.411,-178.643,15.150,150.886
C04857=1108.789,385.741,-90.375,-178.645,15.147,150.886
C04858=1108.784,385.494,-90.339,-178.648,15.142,150.885
C04859=1108.779,385.247,-90.302,-178.651,15.138,150.885
C04860=1108.773,385.000,-90.265,-178.653,15.134,150.884
C04861=1108.768,384.753,-90.228,-178.656,15.130,150.884
C04862=1108.762,384.505,-90.193,-178.658,15.126,150.883
C04863=1108.757,384.259,-90.156,-178.661,15.122,150.883
C04864=1108.747,383.847,-90.095,-178.665,15.115,150.882
C04865=1108.738,383.435,-90.034,-178.669,15.108,150.881
C04866=1108.729,383.023,-89.973,-178.673,15.101,150.881
C04867=1108.719,382.612,-89.913,-178.678,15.094,150.880
C04868=1108.713,382.364,-89.877,-178.680,15.091,150.879
C04869=1108.708,382.117,-89.840,-178.683,15.086,150.879
C04870=1108.702,381.870,-89.804,-178.685,15.083,150.879
C04871=1108.696,381.623,-89.768,-178.688,15.079,150.878
C04872=1108.691,381.376,-89.732,-178.691,15.074,150.878
C04873=1108.685,381.128,-89.696,-178.693,15.071,150.877
C04874=1108.679,380.881,-89.659,-178.696,15.067,150.877
C04875=1108.674,380.634,-89.623,-178.699,15.063,150.877
C04876=1108.667,380.387,-89.587,-178.702,15.059,150.876
C04877=1108.663,380.140,-89.551,-178.704,15.055,150.876
C04878=1108.656,379.893,-89.515,-178.707,15.051,150.875
C04879=1108.650,379.645,-89.479,-178.709,15.048,150.875
C04880=1108.645,379.398,-89.442,-178.712,15.044,150.875
C04881=1108.639,379.151,-89.406,-178.715,15.040,150.874
C04882=1108.634,378.903,-89.369,-178.717,15.036,150.874
C04883=1108.628,378.656,-89.334,-178.720,15.032,150.873
C04884=1108.622,378.409,-89.298,-178.723,15.029,150.873
C04885=1108.617,378.162,-89.262,-178.725,15.025,150.873
C04886=1108.611,377.914,-89.226,-178.728,15.021,150.872
C04887=1108.606,377.667,-89.190,-178.731,15.018,150.872
C04888=1108.600,377.420,-89.153,-178.734,15.013,150.872
C04889=1108.594,377.172,-89.118,-178.736,15.010,150.871
C04890=1108.589,376.925,-89.082,-178.739,15.006,150.871
C04891=1108.583,376.678,-89.047,-178.741,15.002,150.871
C04892=1108.578,376.431,-89.010,-178.745,14.999,150.870
C04893=1108.571,376.183,-88.974,-178.747,14.995,150.870
C04894=1108.566,375.936,-88.939,-178.750,14.991,150.870
C04895=1108.561,375.688,-88.903,-178.752,14.988,150.869
C04896=1108.555,375.442,-88.866,-178.756,14.984,150.869
C04897=1108.549,375.194,-88.831,-178.758,14.980,150.869
C04898=1108.544,374.947,-88.795,-178.761,14.977,150.869
C04899=1108.538,374.699,-88.759,-178.764,14.973,150.868
C04900=1108.533,374.452,-88.724,-178.766,14.970,150.868
C04901=1108.527,374.205,-88.688,-178.769,14.966,150.868
C04902=1108.521,373.958,-88.653,-178.772,14.963,150.867
C04903=1108.515,373.711,-88.616,-178.775,14.959,150.867
C04904=1108.510,373.464,-88.581,-178.778,14.956,150.867
C04905=1108.504,373.216,-88.545,-178.780,14.952,150.867
C04906=1108.498,372.969,-88.510,-178.784,14.949,150.867
C04907=1108.492,372.721,-88.474,-178.786,14.945,150.866
C04908=1108.487,372.474,-88.439,-178.789,14.941,150.866
C04909=1108.481,372.226,-88.402,-178.792,14.938,150.866
C04910=1108.476,371.979,-88.367,-178.794,14.935,150.865
C04911=1108.470,371.732,-88.331,-178.797,14.931,150.865
C04912=1108.465,371.485,-88.296,-178.800,14.928,150.865
C04913=1108.458,371.237,-88.260,-178.803,14.925,150.865
C04914=1108.453,370.990,-88.225,-178.806,14.921,150.865
C04915=1108.447,370.742,-88.189,-178.809,14.918,150.864
C04916=1108.439,370.357,-88.134,-178.813,14.913,150.864
C04917=1108.430,369.972,-88.079,-178.818,14.907,150.864
C04918=1108.420,369.587,-88.024,-178.822,14.903,150.863
C04919=1108.412,369.202,-87.969,-178.826,14.897,150.863
C04920=1108.407,368.955,-87.934,-178.829,14.894,150.863
C04921=1108.400,368.707,-87.899,-178.832,14.890,150.863
C04922=1108.395,368.460,-87.863,-178.835,14.887,150.863
C04923=1108.389,368.212,-87.827,-178.838,14.884,150.862
C04924=1108.384,367.966,-87.792,-178.841,14.880,150.862
C04925=1108.378,367.718,-87.757,-178.844,14.878,150.862
C04926=1108.372,367.470,-87.722,-178.846,14.874,150.862
C04927=1108.367,367.223,-87.686,-178.850,14.871,150.862
C04928=1108.361,366.975,-87.651,-178.853,14.868,150.862
C04929=1108.356,366.728,-87.616,-178.855,14.865,150.862
C04930=1108.350,366.481,-87.581,-178.859,14.861,150.861
C04931=1108.345,366.233,-87.546,-178.861,14.858,150.861
C04932=1108.339,365.986,-87.511,-178.864,14.855,150.861
C04933=1108.333,365.739,-87.475,-178.867,14.852,150.861
C04934=1108.327,365.491,-87.440,-178.870,14.849,150.861
C04935=1108.322,365.244,-87.405,-178.873,14.846,150.861
C04936=1108.316,364.996,-87.370,-178.876,14.843,150.861
C04937=1108.310,364.749,-87.335,-178.879,14.840,150.860
C04938=1108.305,364.501,-87.301,-178.882,14.836,150.860
C04939=1108.299,364.254,-87.265,-178.885,14.833,150.860
C04940=1108.294,364.006,-87.230,-178.888,14.831,150.860
C04941=1108.288,363.759,-87.196,-178.891,14.828,150.860
C04942=1108.282,363.511,-87.160,-178.894,14.824,150.860
C04943=1108.276,363.264,-87.125,-178.897,14.821,150.860
C04944=1108.271,363.016,-87.090,-178.900,14.818,150.860
C04945=1108.265,362.769,-87.055,-178.903,14.816,150.860
C04946=1108.259,362.522,-87.021,-178.906,14.812,150.860
C04947=1108.254,362.275,-86.985,-178.909,14.809,150.860
C04948=1108.248,362.027,-86.951,-178.912,14.807,150.860
C04949=1108.242,361.779,-86.916,-178.915,14.804,150.860
C04950=1108.237,361.532,-86.881,-178.918,14.801,150.859
C04951=1108.231,361.284,-86.846,-178.921,14.798,150.859
C04952=1108.225,361.036,-86.812,-178.924,14.795,150.859
C04953=1108.220,360.789,-86.776,-178.927,14.792,150.859
C04954=1108.214,360.542,-86.742,-178.930,14.789,150.859
C04955=1108.208,360.294,-86.707,-178.933,14.786,150.859
C04956=1108.202,360.047,-86.673,-178.937,14.783,150.859
C04957=1108.197,359.800,-86.638,-178.939,14.780,150.859
C04958=1108.191,359.551,-86.603,-178.943,14.778,150.859
C04959=1108.186,359.304,-86.569,-178.946,14.775,150.859
C04960=1108.180,359.057,-86.534,-178.948,14.772,150.859
C04961=1108.174,358.810,-86.500,-178.951,14.769,150.859
C04962=1108.169,358.561,-86.464,-178.955,14.767,150.859
C04963=1108.163,358.314,-86.430,-178.958,14.763,150.859
C04964=1108.158,358.067,-86.396,-178.961,14.761,150.859
C04965=1108.152,357.819,-86.362,-178.964,14.758,150.859
C04966=1108.146,357.572,-86.326,-178.967,14.755,150.859
C04967=1108.140,357.324,-86.292,-178.970,14.753,150.859
C04968=1108.132,356.954,-86.240,-178.975,14.749,150.859
C04969=1108.123,356.584,-86.189,-178.980,14.744,150.859
C04970=1108.115,356.214,-86.138,-178.984,14.740,150.859
C04971=1108.107,355.843,-86.086,-178.989,14.736,150.859
C04972=1108.101,355.595,-86.052,-178.992,14.734,150.859
C04973=1108.095,355.348,-86.018,-178.995,14.731,150.859
C04974=1108.089,355.100,-85.983,-178.998,14.728,150.859
C04975=1108.083,354.853,-85.949,-179.001,14.726,150.859
C04976=1108.078,354.605,-85.914,-179.004,14.723,150.859
C04977=1108.072,354.358,-85.880,-179.008,14.720,150.859
C04978=1108.067,354.110,-85.845,-179.011,14.718,150.860
C04979=1108.061,353.863,-85.811,-179.014,14.715,150.859
C04980=1108.055,353.615,-85.777,-179.017,14.712,150.860
C04981=1108.050,353.367,-85.742,-179.020,14.710,150.860
C04982=1108.044,353.119,-85.709,-179.023,14.707,150.860
C04983=1108.038,352.872,-85.675,-179.027,14.705,150.860
C04984=1108.033,352.624,-85.640,-179.030,14.702,150.860
C04985=1108.027,352.377,-85.606,-179.033,14.700,150.860
C04986=1108.021,352.129,-85.572,-179.036,14.697,150.860
C04987=1108.015,351.882,-85.538,-179.039,14.695,150.860
C04988=1108.010,351.634,-85.504,-179.042,14.692,150.860
C04989=1108.004,351.386,-85.470,-179.045,14.690,150.860
C04990=1107.999,351.139,-85.436,-179.049,14.688,150.860
C04991=1107.993,350.892,-85.401,-179.052,14.685,150.861
C04992=1107.988,350.644,-85.368,-179.055,14.683,150.861
C04993=1107.982,350.396,-85.333,-179.058,14.680,150.861
C04994=1107.976,350.148,-85.299,-179.061,14.678,150.861
C04995=1107.970,349.900,-85.266,-179.065,14.674,150.861
C04996=1107.965,349.653,-85.231,-179.068,14.672,150.861
C04997=1107.959,349.406,-85.197,-179.072,14.670,150.861
C04998=1107.953,349.158,-85.164,-179.075,14.667,150.861
C04999=1107.948,348.910,-85.130,-179.078,14.665,150.861
C05000=1107.942,348.663,-85.096,-179.081,14.662,150.861
C05001=1107.936,348.415,-85.062,-179.084,14.660,150.862
C05002=1107.931,348.168,-85.028,-179.088,14.658,150.862
C05003=1107.926,347.920,-84.994,-179.091,14.656,150.862
C05004=1107.920,347.672,-84.960,-179.094,14.653,150.862
C05005=1107.914,347.425,-84.927,-179.098,14.651,150.862
C05006=1107.908,347.177,-84.893,-179.101,14.648,150.862
C05007=1107.903,346.929,-84.859,-179.104,14.646,150.862
C05008=1107.897,346.682,-84.825,-179.107,14.644,150.863
C05009=1107.891,346.433,-84.792,-179.110,14.641,150.863
C05010=1107.885,346.186,-84.758,-179.113,14.640,150.863
C05011=1107.880,345.938,-84.724,-179.116,14.637,150.863
C05012=1107.874,345.691,-84.690,-179.120,14.635,150.863
C05013=1107.869,345.443,-84.656,-179.123,14.633,150.863
C05014=1107.863,345.195,-84.622,-179.126,14.631,150.864
C05015=1107.857,344.948,-84.589,-179.130,14.628,150.864
C05016=1107.852,344.700,-84.556,-179.133,14.626,150.864
C05017=1107.846,344.452,-84.522,-179.136,14.624,150.864
C05018=1107.840,344.204,-84.488,-179.140,14.621,150.864
C05019=1107.835,343.957,-84.455,-179.143,14.619,150.865
C05020=1107.826,343.589,-84.405,-179.148,14.616,150.865
C05021=1107.818,343.221,-84.355,-179.153,14.612,150.865
C05022=1107.809,342.853,-84.306,-179.158,14.609,150.865
C05023=1107.801,342.485,-84.256,-179.162,14.606,150.866
C05024=1107.795,342.237,-84.223,-179.166,14.604,150.866
C05025=1107.789,341.989,-84.189,-179.169,14.602,150.866
C05026=1107.784,341.741,-84.155,-179.173,14.600,150.866
C05027=1107.778,341.494,-84.122,-179.176,14.597,150.867
C05028=1107.772,341.246,-84.089,-179.179,14.595,150.867
C05029=1107.766,340.998,-84.056,-179.183,14.593,150.867
C05030=1107.761,340.750,-84.023,-179.186,14.591,150.867
C05031=1107.755,340.503,-83.988,-179.190,14.589,150.868
C05032=1107.749,340.255,-83.955,-179.192,14.587,150.868
C05033=1107.744,340.008,-83.922,-179.196,14.585,150.868
C05034=1107.739,339.760,-83.889,-179.199,14.583,150.868
C05035=1107.733,339.512,-83.856,-179.202,14.581,150.868
C05036=1107.727,339.264,-83.823,-179.206,14.579,150.869
C05037=1107.721,339.016,-83.789,-179.209,14.576,150.869
C05038=1107.716,338.769,-83.756,-179.213,14.574,150.869
C05039=1107.710,338.521,-83.723,-179.216,14.572,150.870
C05040=1107.704,338.273,-83.690,-179.219,14.571,150.870
C05041=1107.699,338.025,-83.657,-179.223,14.569,150.870
C05042=1107.693,337.777,-83.623,-179.226,14.567,150.870
C05043=1107.687,337.530,-83.591,-179.229,14.565,150.871
C05044=1107.682,337.282,-83.558,-179.233,14.563,150.871
C05045=1107.676,337.035,-83.524,-179.237,14.561,150.871
C05046=1107.670,336.787,-83.492,-179.239,14.559,150.871
C05047=1107.664,336.539,-83.458,-179.243,14.557,150.872
C05048=1107.659,336.291,-83.425,-179.246,14.555,150.872
C05049=1107.652,336.044,-83.392,-179.250,14.553,150.872
C05050=1107.647,335.795,-83.359,-179.253,14.551,150.872
C05051=1107.642,335.548,-83.327,-179.257,14.549,150.873
C05052=1107.636,335.300,-83.294,-179.260,14.548,150.873
C05053=1107.630,335.052,-83.260,-179.263,14.546,150.873
C05054=1107.625,334.804,-83.227,-179.267,14.544,150.874
C05055=1107.619,334.557,-83.194,-179.270,14.541,150.874
C05056=1107.613,334.308,-83.162,-179.274,14.539,150.874
C05057=1107.608,334.061,-83.129,-179.277,14.538,150.875
C05058=1107.602,333.813,-83.096,-179.280,14.536,150.875
C05059=1107.597,333.566,-83.063,-179.284,14.534,150.875
C05060=1107.591,333.317,-83.031,-179.287,14.532,150.876
C05061=1107.586,333.070,-82.998,-179.291,14.530,150.876
C05062=1107.579,332.823,-82.965,-179.294,14.529,150.876
C05063=1107.574,332.574,-82.932,-179.298,14.527,150.877
C05064=1107.568,332.326,-82.899,-179.301,14.525,150.877
C05065=1107.562,332.079,-82.866,-179.305,14.523,150.877
C05066=1107.557,331.831,-82.835,-179.307,14.522,150.878
C05067=1107.551,331.583,-82.801,-179.311,14.520,150.878
C05068=1107.545,331.336,-82.769,-179.315,14.518,150.878
C05069=1107.540,331.087,-82.736,-179.318,14.516,150.879
C05070=1107.533,330.839,-82.703,-179.321,14.515,150.879
C05071=1107.528,330.592,-82.671,-179.325,14.513,150.879
C05072=1107.519,330.217,-82.622,-179.330,14.510,150.880
C05073=1107.510,329.843,-82.573,-179.335,14.508,150.880
C05074=1107.502,329.469,-82.524,-179.341,14.505,150.881
C05075=1107.493,329.094,-82.475,-179.346,14.503,150.882
C05076=1107.487,328.847,-82.441,-179.349,14.501,150.882
C05077=1107.482,328.599,-82.410,-179.353,14.500,150.882
C05078=1107.476,328.351,-82.377,-179.357,14.498,150.883
C05079=1107.470,328.103,-82.345,-179.360,14.497,150.883
C05080=1107.464,327.855,-82.311,-179.363,14.495,150.883
C05081=1107.459,327.608,-82.280,-179.367,14.493,150.884
C05082=1107.453,327.360,-82.248,-179.371,14.491,150.884
C05083=1107.447,327.112,-82.214,-179.374,14.490,150.885
C05084=1107.442,326.864,-82.183,-179.378,14.488,150.885
C05085=1107.436,326.617,-82.150,-179.381,14.486,150.885
C05086=1107.430,326.368,-82.118,-179.384,14.485,150.886
C05087=1107.424,326.120,-82.085,-179.388,14.483,150.886
C05088=1107.419,325.873,-82.053,-179.392,14.482,150.887
C05089=1107.413,325.625,-82.021,-179.395,14.480,150.887
C05090=1107.407,325.377,-81.989,-179.398,14.479,150.887
C05091=1107.402,325.129,-81.957,-179.402,14.477,150.888
C05092=1107.396,324.881,-81.924,-179.405,14.476,150.888
C05093=1107.390,324.634,-81.892,-179.409,14.474,150.889
C05094=1107.384,324.385,-81.860,-179.413,14.472,150.889
C05095=1107.378,324.137,-81.828,-179.416,14.471,150.889
C05096=1107.373,323.890,-81.795,-179.419,14.469,150.890
C05097=1107.367,323.642,-81.763,-179.423,14.468,150.890
C05098=1107.361,323.394,-81.731,-179.426,14.467,150.891
C05099=1107.356,323.146,-81.700,-179.430,14.465,150.891
C05100=1107.350,322.898,-81.668,-179.434,14.463,150.892
C05101=1107.345,322.650,-81.636,-179.437,14.462,150.892
C05102=1107.339,322.402,-81.603,-179.440,14.460,150.892
C05103=1107.334,322.155,-81.571,-179.444,14.459,150.893
C05104=1107.328,321.907,-81.539,-179.447,14.457,150.893
C05105=1107.322,321.658,-81.507,-179.451,14.456,150.894
C05106=1107.316,321.411,-81.475,-179.455,14.454,150.894
C05107=1107.310,321.163,-81.443,-179.458,14.453,150.895
C05108=1107.305,320.915,-81.411,-179.462,14.451,150.895
C05109=1107.299,320.667,-81.379,-179.465,14.450,150.895
C05110=1107.294,320.419,-81.348,-179.469,14.449,150.896
C05111=1107.288,320.171,-81.315,-179.472,14.447,150.896
C05112=1107.283,319.923,-81.284,-179.475,14.446,150.897
C05113=1107.277,319.675,-81.252,-179.479,14.444,150.897
C05114=1107.272,319.428,-81.220,-179.483,14.442,150.898
C05115=1107.266,319.180,-81.188,-179.486,14.441,150.898
C05116=1107.260,318.932,-81.156,-179.490,14.440,150.898
C05117=1107.254,318.684,-81.124,-179.493,14.439,150.899
C05118=1107.249,318.436,-81.093,-179.497,14.437,150.899
C05119=1107.244,318.188,-81.062,-179.501,14.435,150.900
C05120=1107.238,317.940,-81.029,-179.504,14.434,150.900
C05121=1107.232,317.692,-80.998,-179.508,14.433,150.901
C05122=1107.226,317.444,-80.966,-179.511,14.432,150.901
C05123=1107.221,317.197,-80.934,-179.515,14.430,150.902
C05124=1107.212,316.815,-80.885,-179.520,14.427,150.902
C05125=1107.204,316.434,-80.837,-179.526,14.426,150.903
C05126=1107.196,316.053,-80.789,-179.531,14.423,150.904
C05127=1107.187,315.671,-80.740,-179.537,14.422,150.905
C05128=1107.181,315.423,-80.708,-179.541,14.420,150.905
C05129=1107.175,315.175,-80.676,-179.544,14.419,150.906
C05130=1107.170,314.927,-80.645,-179.548,14.418,150.906
C05131=1107.164,314.679,-80.614,-179.551,14.417,150.907
C05132=1107.158,314.431,-80.582,-179.555,14.415,150.907
C05133=1107.152,314.183,-80.550,-179.558,14.414,150.907
C05134=1107.147,313.935,-80.519,-179.562,14.413,150.908
C05135=1107.141,313.688,-80.488,-179.565,14.412,150.909
C05136=1107.135,313.440,-80.456,-179.569,14.411,150.909
C05137=1107.130,313.191,-80.425,-179.573,14.409,150.910
C05138=1107.123,312.944,-80.394,-179.576,14.408,150.910
C05139=1107.118,312.696,-80.362,-179.580,14.407,150.911
C05140=1107.112,312.447,-80.331,-179.584,14.406,150.911
C05141=1107.106,312.200,-80.300,-179.587,14.404,150.912
C05142=1107.101,311.952,-80.269,-179.591,14.403,150.912
C05143=1107.095,311.704,-80.237,-179.595,14.402,150.913
C05144=1107.089,311.456,-80.206,-179.598,14.401,150.913
C05145=1107.083,311.208,-80.174,-179.602,14.400,150.914
C05146=1107.077,310.960,-80.144,-179.605,14.399,150.914
C05147=1107.072,310.712,-80.112,-179.609,14.398,150.915
C05148=1107.066,310.463,-80.081,-179.613,14.397,150.916
C05149=1107.060,310.216,-80.050,-179.616,14.395,150.916
C05150=1107.055,309.968,-80.019,-179.620,14.395,150.917
C05151=1107.048,309.720,-79.988,-179.624,14.393,150.917
C05152=1107.043,309.472,-79.957,-179.627,14.392,150.918
C05153=1107.038,309.225,-79.925,-179.631,14.390,150.918
C05154=1107.031,308.976,-79.894,-179.634,14.390,150.919
C05155=1107.026,308.729,-79.863,-179.638,14.388,150.919
C05156=1107.020,308.481,-79.832,-179.642,14.388,150.920
C05157=1107.015,308.233,-79.801,-179.646,14.386,150.920
C05158=1107.008,307.985,-79.770,-179.649,14.385,150.921
C05159=1107.003,307.737,-79.739,-179.653,14.384,150.922
C05160=1106.998,307.489,-79.709,-179.656,14.383,150.922
C05161=1106.992,307.241,-79.676,-179.660,14.382,150.923
C05162=1106.986,306.992,-79.646,-179.664,14.381,150.923
C05163=1106.981,306.745,-79.615,-179.668,14.380,150.924
C05164=1106.976,306.496,-79.584,-179.671,14.379,150.924
C05165=1106.969,306.249,-79.553,-179.675,14.377,150.925
C05166=1106.963,306.001,-79.522,-179.679,14.377,150.926
C05167=1106.958,305.753,-79.492,-179.682,14.375,150.926
C05168=1106.952,305.505,-79.461,-179.686,14.375,150.927
C05169=1106.947,305.257,-79.430,-179.690,14.373,150.927
C05170=1106.940,305.009,-79.399,-179.693,14.372,150.928
C05171=1106.935,304.761,-79.368,-179.697,14.371,150.928
C05172=1106.929,304.513,-79.337,-179.700,14.370,150.929
C05173=1106.924,304.265,-79.307,-179.705,14.369,150.930
C05174=1106.919,304.017,-79.276,-179.708,14.368,150.930
C05175=1106.913,303.769,-79.245,-179.712,14.367,150.931
C05176=1106.905,303.390,-79.198,-179.717,14.366,150.932
C05177=1106.896,303.012,-79.151,-179.723,14.364,150.932
C05178=1106.887,302.633,-79.104,-179.729,14.362,150.933
C05179=1106.878,302.254,-79.057,-179.734,14.361,150.934
C05180=1106.872,302.006,-79.027,-179.739,14.360,150.935
C05181=1106.867,301.758,-78.996,-179.742,14.359,150.935
C05182=1106.862,301.510,-78.966,-179.745,14.358,150.936
C05183=1106.856,301.262,-78.934,-179.749,14.357,150.937
C05184=1106.850,301.014,-78.904,-179.753,14.356,150.937
C05185=1106.844,300.765,-78.874,-179.757,14.355,150.938
C05186=1106.839,300.517,-78.843,-179.760,14.354,150.938
C05187=1106.834,300.269,-78.813,-179.764,14.353,150.939
C05188=1106.828,300.022,-78.783,-179.767,14.352,150.940
C05189=1106.823,299.773,-78.752,-179.772,14.351,150.940
C05190=1106.817,299.526,-78.721,-179.775,14.350,150.941
C05191=1106.811,299.278,-78.691,-179.778,14.349,150.941
C05192=1106.806,299.030,-78.660,-179.783,14.348,150.942
C05193=1106.800,298.782,-78.630,-179.786,14.347,150.943
C05194=1106.795,298.533,-78.600,-179.790,14.346,150.943
C05195=1106.789,298.286,-78.570,-179.794,14.346,150.944
C05196=1106.784,298.037,-78.539,-179.798,14.344,150.944
C05197=1106.778,297.790,-78.508,-179.801,14.344,150.945
C05198=1106.772,297.542,-78.478,-179.805,14.343,150.946
C05199=1106.767,297.293,-78.448,-179.809,14.342,150.946
C05200=1106.760,297.045,-78.418,-179.812,14.341,150.947
C05201=1106.754,296.797,-78.387,-179.816,14.340,150.948
C05202=1106.749,296.549,-78.357,-179.820,14.339,150.948
C05203=1106.743,296.301,-78.327,-179.823,14.339,150.949
C05204=1106.738,296.053,-78.296,-179.827,14.338,150.950
C05205=1106.732,295.805,-78.266,-179.831,14.337,150.950
C05206=1106.727,295.556,-78.236,-179.835,14.336,150.951
C05207=1106.721,295.308,-78.206,-179.838,14.335,150.952
C05208=1106.715,295.061,-78.176,-179.842,14.335,150.952
C05209=1106.710,294.812,-78.146,-179.846,14.334,150.953
C05210=1106.704,294.564,-78.116,-179.850,14.333,150.954
C05211=1106.698,294.317,-78.085,-179.853,14.333,150.954
C05212=1106.692,294.068,-78.056,-179.857,14.331,150.955
C05213=1106.687,293.820,-78.025,-179.861,14.331,150.956
C05214=1106.681,293.572,-77.996,-179.865,14.330,150.956
C05215=1106.675,293.324,-77.965,-179.868,14.329,150.957
C05216=1106.670,293.076,-77.936,-179.872,14.328,150.957
C05217=1106.664,292.828,-77.905,-179.876,14.327,150.958
C05218=1106.658,292.579,-77.876,-179.880,14.327,150.959
C05219=1106.653,292.332,-77.845,-179.883,14.326,150.959
C05220=1106.647,292.083,-77.816,-179.887,14.325,150.960
C05221=1106.641,291.835,-77.785,-179.891,14.325,150.961
C05222=1106.636,291.587,-77.756,-179.894,14.324,150.961
C05223=1106.630,291.339,-77.726,-179.899,14.323,150.962
C05224=1106.624,291.091,-77.696,-179.902,14.322,150.963
C05225=1106.618,290.843,-77.666,-179.906,14.321,150.964
C05226=1106.612,290.595,-77.636,-179.910,14.321,150.964
C05227=1106.607,290.347,-77.607,-179.914,14.320,150.965
C05228=1106.599,289.982,-77.563,-179.919,14.319,150.966
C05229=1106.590,289.617,-77.519,-179.925,14.318,150.967
C05230=1106.582,289.252,-77.476,-179.930,14.317,150.968
C05231=1106.574,288.888,-77.432,-179.936,14.316,150.969
C05232=1106.568,288.640,-77.402,-179.940,14.316,150.970
C05233=1106.562,288.391,-77.372,-179.943,14.315,150.970
C05234=1106.557,288.143,-77.342,-179.947,14.314,150.971
C05235=1106.551,287.895,-77.313,-179.951,14.314,150.972
C05236=1106.545,287.647,-77.283,-179.954,14.313,150.972
C05237=1106.539,287.399,-77.253,-179.959,14.312,150.973
C05238=1106.534,287.150,-77.224,-179.963,14.312,150.974
C05239=1106.528,286.902,-77.194,-179.966,14.311,150.975
C05240=1106.522,286.654,-77.165,-179.970,14.310,150.975
C05241=1106.517,286.406,-77.135,-179.974,14.310,150.976
C05242=1106.511,286.158,-77.106,-179.977,14.309,150.977
C05243=1106.505,285.910,-77.076,-179.982,14.308,150.977
C05244=1106.500,285.661,-77.047,-179.985,14.308,150.978
C05245=1106.494,285.413,-77.017,-179.989,14.308,150.979
C05246=1106.489,285.165,-76.988,-179.993,14.307,150.980
C05247=1106.482,284.916,-76.959,-179.997,14.306,150.980
C05248=1106.477,284.669,-76.929,180.000,14.305,150.981
C05249=1106.472,284.421,-76.899,179.996,14.305,150.982
C05250=1106.465,284.173,-76.870,179.992,14.304,150.982
C05251=1106.460,283.924,-76.840,179.988,14.304,150.983
C05252=1106.454,283.676,-76.811,179.985,14.303,150.984
C05253=1106.449,283.428,-76.782,179.980,14.302,150.984
C05254=1106.443,283.180,-76.752,179.977,14.302,150.985
C05255=1106.438,282.931,-76.723,179.973,14.302,150.986
C05256=1106.431,282.683,-76.694,179.969,14.301,150.987
C05257=1106.426,282.435,-76.664,179.965,14.300,150.987
C05258=1106.420,282.187,-76.636,179.962,14.300,150.988
C05259=1106.415,281.938,-76.606,179.958,14.299,150.989
C05260=1106.409,281.690,-76.577,179.953,14.298,150.990
C05261=1106.403,281.442,-76.548,179.950,14.298,150.990
C05262=1106.398,281.194,-76.518,179.946,14.297,150.991
C05263=1106.392,280.946,-76.489,179.943,14.297,150.992
C05264=1106.387,280.698,-76.460,179.938,14.296,150.992
C05265=1106.380,280.449,-76.431,179.935,14.296,150.993
C05266=1106.375,280.201,-76.401,179.931,14.296,150.994
C05267=1106.369,279.953,-76.373,179.927,14.295,150.995
C05268=1106.364,279.704,-76.344,179.923,14.294,150.995
C05269=1106.358,279.456,-76.314,179.919,14.294,150.996
C05270=1106.352,279.208,-76.285,179.916,14.294,150.997
C05271=1106.347,278.960,-76.256,179.912,14.293,150.998
C05272=1106.341,278.711,-76.227,179.908,14.292,150.998
C05273=1106.335,278.463,-76.198,179.904,14.292,150.999
C05274=1106.329,278.216,-76.170,179.901,14.291,151.000
C05275=1106.324,277.967,-76.140,179.897,14.291,151.001
C05276=1106.318,277.719,-76.112,179.892,14.290,151.001
C05277=1106.312,277.470,-76.082,179.889,14.290,151.002
C05278=1106.307,277.223,-76.053,179.885,14.290,151.003
C05279=1106.302,276.974,-76.024,179.882,14.289,151.004
C05280=1106.293,276.619,-75.984,179.876,14.289,151.005
C05281=1106.285,276.263,-75.942,179.870,14.288,151.006
C05282=1106.277,275.908,-75.900,179.865,14.287,151.007
C05283=1106.269,275.553,-75.859,179.859,14.287,151.008
C05284=1106.263,275.304,-75.830,179.855,14.286,151.009
C05285=1106.257,275.056,-75.802,179.852,14.286,151.010
C05286=1106.252,274.807,-75.773,179.848,14.286,151.010
C05287=1106.246,274.560,-75.744,179.843,14.285,151.011
C05288=1106.240,274.311,-75.716,179.840,14.285,151.012
C05289=1106.235,274.063,-75.686,179.836,14.284,151.013
C05290=1106.229,273.815,-75.658,179.833,14.284,151.013
C05291=1106.223,273.567,-75.629,179.828,14.283,151.014
C05292=1106.217,273.318,-75.601,179.824,14.283,151.015
C05293=1106.212,273.070,-75.571,179.821,14.283,151.016
C05294=1106.206,272.821,-75.543,179.817,14.282,151.017
C05295=1106.200,272.573,-75.514,179.813,14.282,151.017
C05296=1106.195,272.325,-75.486,179.809,14.281,151.018
C05297=1106.190,272.076,-75.457,179.805,14.281,151.019
C05298=1106.184,271.829,-75.428,179.802,14.281,151.020
C05299=1106.178,271.580,-75.400,179.798,14.281,151.020
C05300=1106.172,271.332,-75.371,179.794,14.280,151.021
C05301=1106.166,271.084,-75.343,179.790,14.280,151.022
C05302=1106.160,270.835,-75.315,179.786,14.279,151.023
C05303=1106.156,270.587,-75.286,179.782,14.279,151.024
C05304=1106.150,270.338,-75.257,179.778,14.279,151.024
C05305=1106.144,270.090,-75.229,179.775,14.279,151.025
C05306=1106.138,269.842,-75.201,179.770,14.278,151.026
C05307=1106.132,269.594,-75.172,179.767,14.277,151.027
C05308=1106.127,269.345,-75.144,179.763,14.277,151.028
C05309=1106.121,269.097,-75.116,179.759,14.277,151.028
C05310=1106.115,268.849,-75.088,179.755,14.277,151.029
C05311=1106.109,268.601,-75.059,179.751,14.277,151.030
C05312=1106.104,268.352,-75.031,179.747,14.276,151.031
C05313=1106.099,268.103,-75.002,179.743,14.276,151.032
C05314=1106.093,267.855,-74.974,179.739,14.276,151.032
C05315=1106.087,267.607,-74.945,179.736,14.275,151.033
C05316=1106.081,267.358,-74.916,179.732,14.275,151.034
C05317=1106.076,267.110,-74.888,179.728,14.275,151.035
C05318=1106.070,266.862,-74.860,179.724,14.274,151.036
C05319=1106.065,266.614,-74.832,179.720,14.274,151.036
C05320=1106.059,266.365,-74.804,179.716,14.274,151.037
C05321=1106.053,266.117,-74.776,179.713,14.274,151.038
C05322=1106.047,265.868,-74.748,179.709,14.274,151.039
C05323=1106.042,265.620,-74.720,179.705,14.274,151.040
C05324=1106.037,265.372,-74.692,179.701,14.273,151.040
C05325=1106.031,265.123,-74.663,179.697,14.272,151.041
C05326=1106.025,264.875,-74.635,179.693,14.272,151.042
C05327=1106.019,264.626,-74.607,179.689,14.272,151.043
C05328=1106.014,264.378,-74.579,179.686,14.272,151.044
C05329=1106.007,264.130,-74.551,179.682,14.272,151.045
C05330=1106.002,263.882,-74.523,179.678,14.272,151.045
C05331=1105.996,263.633,-74.495,179.673,14.271,151.046
C05332=1105.988,263.281,-74.455,179.668,14.271,151.047
C05333=1105.980,262.928,-74.415,179.662,14.270,151.049
C05334=1105.972,262.575,-74.376,179.657,14.270,151.050
C05335=1105.963,262.224,-74.337,179.652,14.271,151.051
C05336=1105.957,261.975,-74.308,179.647,14.270,151.052
C05337=1105.952,261.727,-74.280,179.643,14.270,151.053
C05338=1105.946,261.478,-74.252,179.640,14.269,151.053
C05339=1105.940,261.230,-74.225,179.636,14.269,151.054
C05340=1105.934,260.981,-74.197,179.632,14.269,151.055
C05341=1105.929,260.733,-74.169,179.628,14.269,151.056
C05342=1105.923,260.484,-74.141,179.624,14.269,151.057
C05343=1105.917,260.236,-74.113,179.620,14.269,151.058
C05344=1105.912,259.988,-74.085,179.616,14.269,151.059
C05345=1105.906,259.739,-74.058,179.612,14.268,151.059
C05346=1105.900,259.491,-74.030,179.608,14.268,151.060
C05347=1105.894,259.242,-74.002,179.604,14.268,151.061
C05348=1105.889,258.994,-73.974,179.601,14.268,151.062
C05349=1105.884,258.746,-73.947,179.597,14.268,151.063
C05350=1105.877,258.497,-73.919,179.593,14.268,151.064
C05351=1105.871,258.249,-73.891,179.589,14.268,151.065
C05352=1105.866,258.000,-73.864,179.585,14.268,151.065
C05353=1105.860,257.752,-73.836,179.582,14.268,151.066
C05354=1105.854,257.504,-73.808,179.577,14.267,151.067
C05355=1105.848,257.255,-73.781,179.573,14.267,151.068
C05356=1105.843,257.007,-73.753,179.569,14.267,151.069
C05357=1105.838,256.758,-73.726,179.565,14.267,151.070
C05358=1105.831,256.510,-73.698,179.561,14.267,151.070
C05359=1105.826,256.262,-73.670,179.558,14.267,151.071
C05360=1105.821,256.013,-73.643,179.554,14.267,151.072
C05361=1105.814,255.765,-73.615,179.550,14.267,151.073
C05362=1105.809,255.516,-73.588,179.546,14.267,151.074
C05363=1105.803,255.268,-73.561,179.542,14.267,151.075
C05364=1105.798,255.020,-73.534,179.538,14.267,151.075
C05365=1105.792,254.771,-73.505,179.534,14.266,151.076
C05366=1105.786,254.523,-73.479,179.530,14.266,151.077
C05367=1105.781,254.274,-73.451,179.526,14.266,151.078
C05368=1105.774,254.025,-73.424,179.522,14.266,151.079
C05369=1105.769,253.777,-73.396,179.519,14.266,151.080
C05370=1105.763,253.529,-73.369,179.515,14.266,151.081
C05371=1105.758,253.280,-73.342,179.511,14.266,151.081
C05372=1105.752,253.032,-73.313,179.507,14.266,151.082
C05373=1105.746,252.783,-73.287,179.503,14.266,151.083
C05374=1105.741,252.535,-73.259,179.499,14.266,151.084
C05375=1105.735,252.287,-73.232,179.495,14.266,151.085
C05376=1105.730,252.037,-73.205,179.492,14.266,151.086
C05377=1105.724,251.790,-73.177,179.487,14.265,151.087
C05378=1105.719,251.541,-73.150,179.483,14.265,151.088
C05379=1105.713,251.293,-73.123,179.479,14.265,151.088
C05380=1105.708,251.045,-73.095,179.476,14.265,151.089
C05381=1105.701,250.796,-73.068,179.472,14.265,151.090
C05382=1105.696,250.547,-73.041,179.468,14.265,151.091
C05383=1105.690,250.299,-73.015,179.464,14.265,151.092
C05384=1105.682,249.944,-72.975,179.459,14.265,151.093
C05385=1105.674,249.588,-72.936,179.453,14.264,151.094
C05386=1105.666,249.233,-72.898,179.447,14.264,151.095
C05387=1105.658,248.878,-72.860,179.442,14.264,151.097
C05388=1105.652,248.629,-72.832,179.438,14.264,151.098
C05389=1105.647,248.381,-72.805,179.434,14.264,151.098
C05390=1105.642,248.132,-72.778,179.430,14.264,151.099
C05391=1105.636,247.884,-72.751,179.426,14.264,151.100
C05392=1105.630,247.635,-72.724,179.422,14.264,151.101
C05393=1105.625,247.387,-72.697,179.418,14.264,151.102
C05394=1105.619,247.138,-72.670,179.414,14.264,151.103
C05395=1105.614,246.890,-72.644,179.410,14.264,151.104
C05396=1105.608,246.641,-72.616,179.407,14.264,151.105
C05397=1105.602,246.392,-72.590,179.403,14.264,151.105
C05398=1105.596,246.144,-72.563,179.399,14.264,151.106
C05399=1105.591,245.895,-72.536,179.395,14.264,151.107
C05400=1105.585,245.647,-72.508,179.391,14.264,151.108
C05401=1105.579,245.399,-72.482,179.387,14.264,151.109
C05402=1105.574,245.151,-72.455,179.383,14.264,151.110
C05403=1105.569,244.901,-72.428,179.379,14.264,151.111
C05404=1105.563,244.653,-72.402,179.375,14.264,151.112
C05405=1105.557,244.404,-72.375,179.372,14.264,151.112
C05406=1105.551,244.156,-72.348,179.368,14.264,151.113
C05407=1105.546,243.907,-72.321,179.364,14.264,151.114
C05408=1105.540,243.659,-72.294,179.360,14.264,151.115
C05409=1105.534,243.410,-72.268,179.356,14.264,151.116
C05410=1105.529,243.162,-72.241,179.352,14.264,151.117
C05411=1105.523,242.914,-72.214,179.348,14.265,151.118
C05412=1105.517,242.665,-72.188,179.344,14.265,151.119
C05413=1105.511,242.417,-72.161,179.340,14.265,151.120
C05414=1105.507,242.168,-72.134,179.336,14.265,151.120
C05415=1105.501,241.919,-72.108,179.332,14.265,151.121
C05416=1105.495,241.671,-72.081,179.329,14.265,151.122
C05417=1105.489,241.422,-72.055,179.325,14.265,151.123
C05418=1105.484,241.174,-72.028,179.321,14.265,151.124
C05419=1105.478,240.925,-72.002,179.317,14.265,151.125
C05420=1105.472,240.677,-71.975,179.313,14.265,151.126
